C05485=1164.302,294.931,-71.199,-176.927,8.045,148.667
C05486=1164.298,295.179,-71.230,-176.924,8.049,148.668
C05487=1164.294,295.428,-71.259,-176.921,8.052,148.668
C05488=1164.290,295.675,-71.290,-176.919,8.055,148.668
C05489=1164.285,295.924,-71.320,-176.916,8.058,148.668
C05490=1164.282,296.172,-71.350,-176.914,8.061,148.668
C05491=1164.277,296.420,-71.381,-176.911,8.064,148.668
C05492=1164.273,296.668,-71.410,-176.909,8.067,148.668
C05493=1164.269,296.916,-71.441,-176.906,8.070,148.668
C05494=1164.265,297.164,-71.471,-176.904,8.073,148.668
C05495=1164.260,297.413,-71.501,-176.901,8.076,148.668
C05496=1164.256,297.660,-71.532,-176.898,8.079,148.668
C05497=1164.251,297.908,-71.562,-176.896,8.083,148.668
C05498=1164.247,298.157,-71.592,-176.893,8.086,148.668
C05499=1164.243,298.405,-71.623,-176.891,8.089,148.668
C05500=1164.239,298.653,-71.653,-176.888,8.092,148.668
C05501=1164.234,298.901,-71.683,-176.885,8.095,148.668
C05502=1164.231,299.149,-71.713,-176.883,8.098,148.668
C05503=1164.226,299.397,-71.744,-176.880,8.101,148.668
C05504=1164.223,299.645,-71.775,-176.878,8.104,148.669
C05505=1164.218,299.893,-71.805,-176.875,8.107,148.668
C05506=1164.213,300.142,-71.835,-176.872,8.110,148.668
C05507=1164.209,300.390,-71.866,-176.870,8.114,148.669
C05508=1164.205,300.638,-71.897,-176.867,8.117,148.669
C05509=1164.201,300.886,-71.927,-176.865,8.120,148.669
C05510=1164.197,301.134,-71.958,-176.862,8.123,148.669
C05511=1164.192,301.382,-71.988,-176.860,8.126,148.669
C05512=1164.189,301.630,-72.019,-176.857,8.130,148.669
C05513=1164.184,301.879,-72.049,-176.854,8.133,148.669
C05514=1164.179,302.127,-72.080,-176.852,8.136,148.669
C05515=1164.175,302.374,-72.110,-176.849,8.139,148.669
C05516=1164.171,302.623,-72.141,-176.847,8.142,148.669
C05517=1164.167,302.871,-72.172,-176.844,8.145,148.669
C05518=1164.163,303.119,-72.202,-176.841,8.148,148.669
C05519=1164.158,303.367,-72.233,-176.839,8.152,148.669
C05520=1164.154,303.615,-72.264,-176.836,8.155,148.669
C05521=1164.150,303.863,-72.295,-176.834,8.158,148.670
C05522=1164.146,304.111,-72.325,-176.831,8.161,148.670
C05523=1164.142,304.359,-72.356,-176.829,8.164,148.670
C05524=1164.137,304.607,-72.387,-176.826,8.167,148.670
C05525=1164.133,304.855,-72.417,-176.824,8.170,148.670
C05526=1164.130,305.103,-72.449,-176.821,8.173,148.670
C05527=1164.125,305.351,-72.479,-176.818,8.177,148.670
C05528=1164.120,305.599,-72.510,-176.815,8.180,148.670
C05529=1164.116,305.848,-72.541,-176.813,8.184,148.670
C05530=1164.113,306.095,-72.572,-176.810,8.187,148.670
C05531=1164.108,306.343,-72.602,-176.808,8.190,148.670
C05532=1164.104,306.592,-72.633,-176.805,8.193,148.670
C05533=1164.099,306.840,-72.664,-176.803,8.196,148.670
C05534=1164.095,307.087,-72.696,-176.800,8.199,148.671
C05535=1164.091,307.336,-72.727,-176.797,8.202,148.671
C05536=1164.087,307.584,-72.757,-176.795,8.205,148.671
C05537=1164.083,307.832,-72.788,-176.792,8.208,148.671
C05538=1164.079,308.080,-72.820,-176.790,8.212,148.671
C05539=1164.074,308.328,-72.850,-176.787,8.215,148.671
C05540=1164.070,308.576,-72.881,-176.785,8.219,148.671
C05541=1164.066,308.824,-72.912,-176.782,8.222,148.671
C05542=1164.062,309.072,-72.944,-176.780,8.225,148.671
C05543=1164.057,309.320,-72.975,-176.777,8.228,148.671
C05544=1164.053,309.568,-73.005,-176.774,8.231,148.671
C05545=1164.050,309.816,-73.037,-176.772,8.235,148.672
C05546=1164.045,310.064,-73.068,-176.769,8.238,148.672
C05547=1164.041,310.312,-73.099,-176.767,8.241,148.672
C05548=1164.037,310.560,-73.130,-176.764,8.244,148.672
C05549=1164.033,310.808,-73.161,-176.762,8.248,148.672
C05550=1164.028,311.056,-73.193,-176.759,8.251,148.672
C05551=1164.024,311.304,-73.224,-176.756,8.254,148.672
C05552=1164.020,311.552,-73.255,-176.754,8.257,148.672
C05553=1164.015,311.800,-73.286,-176.751,8.260,148.672
C05554=1164.011,312.048,-73.317,-176.749,8.263,148.672
C05555=1164.007,312.296,-73.349,-176.746,8.267,148.673
C05556=1164.003,312.544,-73.380,-176.744,8.270,148.672
C05557=1163.999,312.792,-73.411,-176.741,8.273,148.673
C05558=1163.995,313.040,-73.443,-176.738,8.277,148.673
C05559=1163.991,313.288,-73.474,-176.736,8.280,148.673
C05560=1163.986,313.565,-73.510,-176.733,8.283,148.673
C05561=1163.981,313.843,-73.544,-176.730,8.287,148.673
C05562=1163.976,314.119,-73.579,-176.728,8.290,148.673
C05563=1163.972,314.397,-73.615,-176.725,8.294,148.673
C05564=1163.967,314.644,-73.646,-176.722,8.298,148.674
C05565=1163.963,314.893,-73.678,-176.719,8.300,148.674
C05566=1163.959,315.140,-73.709,-176.717,8.304,148.674
C05567=1163.955,315.388,-73.741,-176.714,8.308,148.674
C05568=1163.951,315.636,-73.772,-176.712,8.311,148.674
C05569=1163.947,315.884,-73.804,-176.709,8.314,148.674
C05570=1163.943,316.132,-73.835,-176.707,8.317,148.674
C05571=1163.939,316.380,-73.866,-176.704,8.320,148.674
C05572=1163.934,316.629,-73.899,-176.702,8.324,148.674
C05573=1163.930,316.876,-73.930,-176.699,8.327,148.674
C05574=1163.926,317.124,-73.962,-176.696,8.331,148.675
C05575=1163.922,317.373,-73.993,-176.694,8.334,148.675
C05576=1163.918,317.620,-74.025,-176.691,8.337,148.675
C05577=1163.914,317.868,-74.057,-176.689,8.340,148.675
C05578=1163.909,318.116,-74.088,-176.686,8.343,148.675
C05579=1163.905,318.364,-74.120,-176.684,8.347,148.675
C05580=1163.902,318.612,-74.151,-176.682,8.350,148.675
C05581=1163.897,318.860,-74.183,-176.678,8.354,148.675
C05582=1163.893,319.108,-74.215,-176.676,8.357,148.676
C05583=1163.888,319.356,-74.247,-176.673,8.360,148.676
C05584=1163.885,319.604,-74.279,-176.671,8.363,148.676
C05585=1163.881,319.852,-74.311,-176.669,8.367,148.676
C05586=1163.876,320.099,-74.343,-176.666,8.369,148.676
C05587=1163.872,320.347,-74.374,-176.663,8.374,148.676
C05588=1163.868,320.596,-74.406,-176.661,8.377,148.676
C05589=1163.863,320.844,-74.438,-176.658,8.380,148.676
C05590=1163.860,321.092,-74.469,-176.656,8.383,148.677
C05591=1163.856,321.340,-74.501,-176.653,8.386,148.677
C05592=1163.852,321.587,-74.533,-176.651,8.389,148.677
C05593=1163.847,321.835,-74.565,-176.648,8.393,148.677
C05594=1163.843,322.083,-74.597,-176.646,8.397,148.677
C05595=1163.840,322.331,-74.629,-176.643,8.400,148.677
C05596=1163.835,322.578,-74.662,-176.640,8.403,148.677
C05597=1163.831,322.826,-74.694,-176.638,8.406,148.678
C05598=1163.827,323.075,-74.726,-176.635,8.409,148.678
C05599=1163.822,323.322,-74.757,-176.633,8.413,148.678
C05600=1163.819,323.570,-74.789,-176.630,8.417,148.678
C05601=1163.814,323.819,-74.822,-176.628,8.420,148.678
C05602=1163.811,324.067,-74.854,-176.625,8.423,148.678
C05603=1163.806,324.314,-74.886,-176.623,8.426,148.678
C05604=1163.802,324.562,-74.918,-176.621,8.430,148.679
C05605=1163.798,324.810,-74.950,-176.617,8.433,148.679
C05606=1163.794,325.058,-74.983,-176.615,8.437,148.679
C05607=1163.790,325.305,-75.014,-176.613,8.440,148.679
C05608=1163.785,325.554,-75.046,-176.610,8.443,148.679
C05609=1163.782,325.802,-75.078,-176.608,8.446,148.679
C05610=1163.777,326.050,-75.111,-176.605,8.450,148.680
C05611=1163.774,326.298,-75.143,-176.603,8.454,148.680
C05612=1163.769,326.545,-75.175,-176.600,8.457,148.680
C05613=1163.765,326.793,-75.208,-176.598,8.460,148.680
C05614=1163.761,327.041,-75.240,-176.595,8.463,148.680
C05615=1163.757,327.289,-75.272,-176.592,8.467,148.680
C05616=1163.753,327.537,-75.305,-176.590,8.470,148.680
C05617=1163.749,327.784,-75.337,-176.587,8.474,148.681
C05618=1163.744,328.032,-75.369,-176.585,8.477,148.681
C05619=1163.740,328.280,-75.402,-176.583,8.480,148.681
C05620=1163.736,328.528,-75.434,-176.579,8.484,148.681
C05621=1163.732,328.777,-75.467,-176.577,8.487,148.681
C05622=1163.728,329.023,-75.499,-176.575,8.490,148.681
C05623=1163.724,329.272,-75.531,-176.573,8.494,148.682
C05624=1163.720,329.519,-75.564,-176.570,8.497,148.682
C05625=1163.716,329.767,-75.596,-176.567,8.501,148.682
C05626=1163.711,330.016,-75.629,-176.565,8.504,148.682
C05627=1163.708,330.263,-75.661,-176.562,8.507,148.682
C05628=1163.703,330.512,-75.694,-176.560,8.511,148.682
C05629=1163.699,330.759,-75.727,-176.558,8.514,148.683
C05630=1163.695,331.007,-75.758,-176.554,8.518,148.683
C05631=1163.691,331.254,-75.792,-176.552,8.521,148.683
C05632=1163.687,331.502,-75.825,-176.550,8.524,148.683
C05633=1163.683,331.750,-75.857,-176.548,8.528,148.683
C05634=1163.679,331.998,-75.890,-176.545,8.532,148.684
C05635=1163.674,332.246,-75.922,-176.542,8.535,148.684
C05636=1163.670,332.494,-75.955,-176.540,8.538,148.684
C05637=1163.667,332.741,-75.988,-176.537,8.541,148.684
C05638=1163.662,332.990,-76.020,-176.534,8.545,148.684
C05639=1163.658,333.237,-76.054,-176.532,8.549,148.684
C05640=1163.654,333.485,-76.085,-176.530,8.552,148.685
C05641=1163.650,333.732,-76.118,-176.527,8.555,148.685
C05642=1163.646,333.980,-76.151,-176.524,8.559,148.685
C05643=1163.642,334.228,-76.184,-176.522,8.562,148.685
C05644=1163.637,334.476,-76.217,-176.520,8.566,148.685
C05645=1163.634,334.724,-76.249,-176.517,8.569,148.685
C05646=1163.630,334.971,-76.283,-176.515,8.572,148.686
C05647=1163.625,335.220,-76.315,-176.512,8.576,148.686
C05648=1163.621,335.467,-76.348,-176.509,8.579,148.686
C05649=1163.617,335.715,-76.381,-176.507,8.583,148.686
C05650=1163.613,335.963,-76.414,-176.505,8.586,148.686
C05651=1163.609,336.210,-76.447,-176.502,8.590,148.687
C05652=1163.605,336.459,-76.480,-176.500,8.593,148.687
C05653=1163.601,336.706,-76.513,-176.497,8.597,148.687
C05654=1163.597,336.954,-76.546,-176.494,8.601,148.687
C05655=1163.592,337.202,-76.579,-176.492,8.604,148.687
C05656=1163.588,337.450,-76.612,-176.490,8.607,148.688
C05657=1163.585,337.697,-76.645,-176.487,8.610,148.688
C05658=1163.581,337.945,-76.678,-176.484,8.614,148.688
C05659=1163.577,338.192,-76.711,-176.482,8.618,148.688
C05660=1163.572,338.440,-76.744,-176.480,8.621,148.688
C05661=1163.568,338.688,-76.777,-176.477,8.624,148.688
C05662=1163.564,338.936,-76.811,-176.475,8.628,148.689
C05663=1163.560,339.183,-76.844,-176.472,8.632,148.689
C05664=1163.555,339.464,-76.880,-176.469,8.636,148.689
C05665=1163.551,339.743,-76.918,-176.466,8.640,148.689
C05666=1163.546,340.023,-76.956,-176.464,8.643,148.690
C05667=1163.541,340.302,-76.993,-176.461,8.647,148.690
C05668=1163.538,340.551,-77.027,-176.458,8.651,148.690
C05669=1163.534,340.799,-77.060,-176.456,8.655,148.690
C05670=1163.530,341.046,-77.093,-176.454,8.658,148.691
C05671=1163.525,341.294,-77.126,-176.452,8.661,148.691
C05672=1163.522,341.541,-77.160,-176.449,8.665,148.691
C05673=1163.517,341.789,-77.193,-176.446,8.669,148.691
C05674=1163.513,342.037,-77.226,-176.444,8.672,148.691
C05675=1163.509,342.284,-77.259,-176.441,8.676,148.692
C05676=1163.505,342.532,-77.293,-176.439,8.679,148.692
C05677=1163.501,342.780,-77.326,-176.437,8.683,148.692
C05678=1163.497,343.028,-77.361,-176.434,8.687,148.692
C05679=1163.493,343.276,-77.394,-176.431,8.690,148.693
C05680=1163.489,343.523,-77.427,-176.429,8.693,148.693
C05681=1163.484,343.771,-77.460,-176.427,8.697,148.693
C05682=1163.480,344.019,-77.493,-176.424,8.701,148.693
C05683=1163.477,344.266,-77.527,-176.422,8.704,148.693
C05684=1163.472,344.514,-77.560,-176.419,8.707,148.694
C05685=1163.469,344.762,-77.594,-176.417,8.711,148.694
C05686=1163.464,345.009,-77.628,-176.414,8.715,148.694
C05687=1163.460,345.257,-77.661,-176.412,8.718,148.694
C05688=1163.456,345.505,-77.694,-176.409,8.722,148.695
C05689=1163.452,345.752,-77.728,-176.407,8.725,148.695
C05690=1163.448,346.000,-77.762,-176.404,8.729,148.695
C05691=1163.444,346.249,-77.796,-176.402,8.733,148.695
C05692=1163.440,346.496,-77.830,-176.399,8.736,148.696
C05693=1163.436,346.743,-77.863,-176.397,8.739,148.696
C05694=1163.432,346.990,-77.897,-176.394,8.744,148.696
C05695=1163.428,347.239,-77.931,-176.392,8.747,148.696
C05696=1163.424,347.487,-77.964,-176.390,8.750,148.696
C05697=1163.420,347.734,-77.998,-176.387,8.754,148.697
C05698=1163.416,347.982,-78.031,-176.385,8.758,148.697
C05699=1163.411,348.229,-78.065,-176.382,8.761,148.697
C05700=1163.407,348.478,-78.099,-176.380,8.765,148.698
C05701=1163.404,348.725,-78.133,-176.377,8.769,148.698
C05702=1163.399,348.972,-78.166,-176.375,8.772,148.698
C05703=1163.395,349.220,-78.200,-176.372,8.776,148.698
C05704=1163.392,349.468,-78.235,-176.370,8.779,148.698
C05705=1163.388,349.715,-78.268,-176.368,8.783,148.699
C05706=1163.383,349.963,-78.302,-176.365,8.787,148.699
C05707=1163.379,350.211,-78.336,-176.363,8.790,148.699
C05708=1163.376,350.458,-78.370,-176.361,8.794,148.700
C05709=1163.371,350.706,-78.404,-176.358,8.798,148.700
C05710=1163.367,350.954,-78.437,-176.355,8.801,148.700
C05711=1163.363,351.202,-78.472,-176.352,8.805,148.700
C05712=1163.359,351.449,-78.506,-176.350,8.808,148.701
C05713=1163.355,351.696,-78.539,-176.348,8.812,148.701
C05714=1163.351,351.945,-78.574,-176.345,8.816,148.701
C05715=1163.347,352.192,-78.608,-176.343,8.819,148.701
C05716=1163.342,352.440,-78.641,-176.341,8.823,148.702
C05717=1163.339,352.688,-78.676,-176.338,8.827,148.702
C05718=1163.335,352.935,-78.710,-176.336,8.830,148.702
C05719=1163.331,353.182,-78.744,-176.333,8.834,148.703
C05720=1163.327,353.430,-78.778,-176.331,8.838,148.703
C05721=1163.323,353.678,-78.812,-176.329,8.841,148.703
C05722=1163.319,353.926,-78.846,-176.326,8.845,148.703
C05723=1163.315,354.173,-78.881,-176.324,8.849,148.704
C05724=1163.311,354.420,-78.915,-176.322,8.852,148.704
C05725=1163.307,354.668,-78.949,-176.319,8.856,148.704
C05726=1163.303,354.915,-78.983,-176.316,8.859,148.704
C05727=1163.298,355.164,-79.017,-176.314,8.864,148.705
C05728=1163.295,355.411,-79.051,-176.312,8.867,148.705
C05729=1163.290,355.659,-79.086,-176.309,8.870,148.705
C05730=1163.287,355.907,-79.120,-176.307,8.875,148.706
C05731=1163.283,356.154,-79.154,-176.305,8.878,148.706
C05732=1163.279,356.402,-79.189,-176.302,8.882,148.706
C05733=1163.275,356.649,-79.223,-176.299,8.886,148.706
C05734=1163.271,356.896,-79.257,-176.297,8.889,148.707
C05735=1163.267,357.144,-79.292,-176.295,8.893,148.707
C05736=1163.262,357.392,-79.326,-176.292,8.897,148.707
C05737=1163.259,357.640,-79.361,-176.290,8.901,148.708
C05738=1163.255,357.887,-79.395,-176.288,8.904,148.708
C05739=1163.251,358.135,-79.429,-176.285,8.908,148.708
C05740=1163.247,358.382,-79.464,-176.283,8.912,148.709
C05741=1163.243,358.630,-79.499,-176.281,8.915,148.709
C05742=1163.239,358.877,-79.533,-176.278,8.919,148.709
C05743=1163.235,359.125,-79.568,-176.275,8.923,148.709
C05744=1163.231,359.372,-79.602,-176.273,8.927,148.710
C05745=1163.228,359.620,-79.637,-176.271,8.930,148.710
C05746=1163.223,359.868,-79.671,-176.268,8.934,148.710
C05747=1163.219,360.116,-79.706,-176.266,8.938,148.711
C05748=1163.215,360.363,-79.740,-176.263,8.942,148.711
C05749=1163.212,360.610,-79.775,-176.261,8.945,148.711
C05750=1163.207,360.858,-79.810,-176.258,8.950,148.712
C05751=1163.204,361.106,-79.844,-176.256,8.953,148.712
C05752=1163.199,361.353,-79.879,-176.254,8.958,148.712
C05753=1163.196,361.601,-79.914,-176.251,8.961,148.713
C05754=1163.191,361.848,-79.949,-176.249,8.964,148.713
C05755=1163.188,362.096,-79.983,-176.247,8.969,148.713
C05756=1163.183,362.343,-80.018,-176.244,8.972,148.714
C05757=1163.180,362.591,-80.053,-176.242,8.976,148.714
C05758=1163.176,362.839,-80.088,-176.240,8.980,148.714
C05759=1163.172,363.085,-80.122,-176.237,8.984,148.715
C05760=1163.168,363.333,-80.157,-176.235,8.987,148.715
C05761=1163.163,363.581,-80.192,-176.232,8.992,148.715
C05762=1163.160,363.828,-80.227,-176.230,8.995,148.716
C05763=1163.156,364.077,-80.262,-176.228,8.999,148.716
C05764=1163.152,364.324,-80.296,-176.226,9.003,148.717
C05765=1163.148,364.571,-80.331,-176.224,9.006,148.717
C05766=1163.144,364.819,-80.366,-176.221,9.011,148.717
C05767=1163.140,365.066,-80.401,-176.219,9.014,148.717
C05768=1163.136,365.348,-80.441,-176.216,9.018,148.718
C05769=1163.132,365.631,-80.481,-176.214,9.023,148.718
C05770=1163.127,365.913,-80.521,-176.211,9.028,148.719
C05771=1163.122,366.196,-80.561,-176.208,9.033,148.719
C05772=1163.118,366.444,-80.596,-176.206,9.036,148.720
C05773=1163.114,366.691,-80.631,-176.204,9.039,148.720
C05774=1163.110,366.939,-80.666,-176.202,9.044,148.721
C05775=1163.106,367.186,-80.702,-176.200,9.047,148.721
C05776=1163.102,367.434,-80.736,-176.197,9.052,148.721
C05777=1163.098,367.681,-80.772,-176.195,9.055,148.722
C05778=1163.095,367.929,-80.807,-176.193,9.059,148.722
C05779=1163.090,368.176,-80.842,-176.191,9.063,148.723
C05780=1163.086,368.424,-80.877,-176.189,9.067,148.723
C05781=1163.082,368.672,-80.912,-176.187,9.070,148.723
C05782=1163.078,368.919,-80.947,-176.185,9.075,148.724
C05783=1163.074,369.166,-80.983,-176.183,9.078,148.724
C05784=1163.071,369.414,-81.018,-176.181,9.082,148.725
C05785=1163.066,369.661,-81.053,-176.179,9.086,148.725
C05786=1163.062,369.908,-81.088,-176.177,9.090,148.726
C05787=1163.059,370.156,-81.124,-176.175,9.094,148.726
C05788=1163.055,370.404,-81.159,-176.172,9.098,148.727
C05789=1163.051,370.651,-81.194,-176.171,9.102,148.727
C05790=1163.047,370.898,-81.229,-176.169,9.106,148.728
C05791=1163.043,371.146,-81.265,-176.167,9.109,148.728
C05792=1163.039,371.393,-81.300,-176.165,9.114,148.729
C05793=1163.035,371.641,-81.335,-176.163,9.117,148.729
C05794=1163.031,371.888,-81.371,-176.161,9.121,148.730
C05795=1163.028,372.136,-81.406,-176.160,9.125,148.730
C05796=1163.023,372.383,-81.441,-176.157,9.129,148.730
C05797=1163.020,372.630,-81.477,-176.156,9.133,148.731
C05798=1163.016,372.878,-81.512,-176.154,9.137,148.732
C05799=1163.012,373.125,-81.549,-176.152,9.140,148.732
C05800=1163.008,373.373,-81.584,-176.151,9.144,148.733
C05801=1163.003,373.620,-81.619,-176.149,9.148,148.733
C05802=1163.000,373.868,-81.654,-176.147,9.152,148.734
C05803=1162.996,374.115,-81.690,-176.146,9.155,148.734
C05804=1162.992,374.363,-81.725,-176.143,9.160,148.735
C05805=1162.987,374.610,-81.761,-176.142,9.164,148.735
C05806=1162.984,374.857,-81.797,-176.140,9.167,148.736
C05807=1162.980,375.105,-81.832,-176.139,9.171,148.736
C05808=1162.977,375.352,-81.868,-176.137,9.175,148.737
C05809=1162.973,375.600,-81.903,-176.136,9.179,148.738
C05810=1162.969,375.847,-81.939,-176.134,9.183,148.738
C05811=1162.964,376.095,-81.975,-176.132,9.187,148.739
C05812=1162.961,376.342,-82.010,-176.131,9.190,148.739
C05813=1162.957,376.589,-82.046,-176.130,9.194,148.740
C05814=1162.953,376.836,-82.082,-176.129,9.197,148.741
C05815=1162.949,377.084,-82.118,-176.127,9.201,148.741
C05816=1162.945,377.332,-82.154,-176.126,9.205,148.742
C05817=1162.941,377.579,-82.189,-176.124,9.209,148.742
C05818=1162.938,377.826,-82.224,-176.123,9.213,148.743
C05819=1162.933,378.074,-82.260,-176.122,9.217,148.744
C05820=1162.929,378.321,-82.296,-176.121,9.220,148.744
C05821=1162.926,378.569,-82.332,-176.119,9.224,148.745
C05822=1162.922,378.816,-82.368,-176.118,9.228,148.745
C05823=1162.918,379.064,-82.404,-176.117,9.232,148.746
C05824=1162.914,379.310,-82.439,-176.116,9.235,148.747
C05825=1162.909,379.558,-82.475,-176.114,9.239,148.747
C05826=1162.906,379.806,-82.511,-176.113,9.243,148.748
C05827=1162.902,380.053,-82.547,-176.113,9.246,148.749
C05828=1162.899,380.300,-82.583,-176.111,9.250,148.750
C05829=1162.894,380.548,-82.619,-176.111,9.254,148.750
C05830=1162.891,380.795,-82.654,-176.109,9.258,148.751
C05831=1162.887,381.043,-82.691,-176.108,9.261,148.751
C05832=1162.882,381.289,-82.726,-176.107,9.265,148.752
C05833=1162.879,381.537,-82.762,-176.107,9.268,148.753
C05834=1162.874,381.785,-82.798,-176.106,9.272,148.754
C05835=1162.871,382.032,-82.834,-176.105,9.276,148.754
C05836=1162.867,382.279,-82.870,-176.104,9.279,148.755
C05837=1162.863,382.527,-82.906,-176.103,9.283,148.756
C05838=1162.859,382.774,-82.942,-176.103,9.286,148.757
C05839=1162.855,383.022,-82.978,-176.102,9.289,148.757
C05840=1162.851,383.269,-83.014,-176.101,9.293,148.758
C05841=1162.848,383.516,-83.050,-176.100,9.297,148.759
C05842=1162.844,383.764,-83.086,-176.100,9.300,148.760
C05843=1162.840,384.011,-83.122,-176.099,9.303,148.760
C05844=1162.836,384.258,-83.159,-176.099,9.307,148.761
C05845=1162.832,384.506,-83.194,-176.098,9.311,148.762
C05846=1162.828,384.753,-83.230,-176.097,9.314,148.762
C05847=1162.824,385.000,-83.266,-176.097,9.318,148.763
C05848=1162.820,385.247,-83.302,-176.096,9.321,148.764
C05849=1162.816,385.495,-83.339,-176.096,9.325,148.765
C05850=1162.812,385.742,-83.374,-176.096,9.328,148.766
C05851=1162.808,385.990,-83.410,-176.096,9.330,148.766
C05852=1162.805,386.237,-83.447,-176.095,9.334,148.767
C05853=1162.800,386.485,-83.483,-176.095,9.337,148.768
C05854=1162.797,386.731,-83.519,-176.094,9.341,148.769
C05855=1162.793,386.979,-83.555,-176.094,9.344,148.769
C05856=1162.789,387.226,-83.592,-176.094,9.347,148.770
C05857=1162.785,387.474,-83.627,-176.094,9.350,148.771
C05858=1162.781,387.721,-83.664,-176.094,9.354,148.772
C05859=1162.778,387.968,-83.699,-176.094,9.356,148.772
C05860=1162.774,388.216,-83.736,-176.094,9.360,148.773
C05861=1162.770,388.463,-83.772,-176.094,9.362,148.774
C05862=1162.766,388.710,-83.809,-176.093,9.366,148.775
C05863=1162.762,388.958,-83.844,-176.094,9.368,148.776
C05864=1162.758,389.205,-83.881,-176.094,9.372,148.777
C05865=1162.754,389.452,-83.917,-176.094,9.375,148.777
C05866=1162.750,389.700,-83.954,-176.094,9.377,148.778
C05867=1162.747,389.947,-83.989,-176.094,9.381,148.779
C05868=1162.743,390.194,-84.026,-176.094,9.384,148.780
C05869=1162.739,390.442,-84.062,-176.094,9.386,148.780
C05870=1162.735,390.689,-84.098,-176.094,9.390,148.781
C05871=1162.731,390.937,-84.134,-176.094,9.392,148.782
C05872=1162.726,391.222,-84.177,-176.095,9.395,148.783
C05873=1162.722,391.508,-84.218,-176.095,9.399,148.784
C05874=1162.718,391.793,-84.260,-176.095,9.402,148.785
C05875=1162.713,392.078,-84.302,-176.095,9.406,148.786
C05876=1162.709,392.325,-84.338,-176.095,9.408,148.787
C05877=1162.705,392.574,-84.375,-176.096,9.411,148.787
C05878=1162.702,392.820,-84.411,-176.096,9.414,148.788
C05879=1162.698,393.068,-84.447,-176.096,9.416,148.789
C05880=1162.694,393.315,-84.483,-176.097,9.419,148.790
C05881=1162.690,393.562,-84.520,-176.097,9.422,148.790
C05882=1162.687,393.810,-84.556,-176.097,9.424,148.791
C05883=1162.683,394.057,-84.592,-176.098,9.427,148.792
C05884=1162.678,394.305,-84.629,-176.098,9.429,148.793
C05885=1162.675,394.552,-84.665,-176.099,9.432,148.794
C05886=1162.671,394.799,-84.702,-176.099,9.434,148.794
C05887=1162.667,395.046,-84.737,-176.100,9.437,148.795
C05888=1162.663,395.294,-84.774,-176.100,9.440,148.796
C05889=1162.659,395.541,-84.810,-176.100,9.441,148.797
C05890=1162.655,395.788,-84.847,-176.101,9.444,148.798
C05891=1162.651,396.035,-84.883,-176.101,9.447,148.798
C05892=1162.647,396.283,-84.919,-176.101,9.449,148.799
C05893=1162.643,396.530,-84.956,-176.102,9.451,148.800
C05894=1162.640,396.778,-84.991,-176.103,9.454,148.801
C05895=1162.636,397.025,-85.028,-176.104,9.456,148.801
C05896=1162.632,397.272,-85.064,-176.104,9.459,148.802
C05897=1162.628,397.520,-85.101,-176.104,9.461,148.803
C05898=1162.624,397.767,-85.137,-176.105,9.463,148.804
C05899=1162.620,398.014,-85.174,-176.105,9.466,148.804
C05900=1162.616,398.261,-85.210,-176.106,9.468,148.805
C05901=1162.613,398.508,-85.246,-176.107,9.470,148.806
C05902=1162.608,398.755,-85.283,-176.107,9.472,148.807
C05903=1162.604,399.003,-85.319,-176.107,9.475,148.807
C05904=1162.601,399.250,-85.355,-176.108,9.477,148.808
C05905=1162.597,399.497,-85.392,-176.109,9.479,148.809
C05906=1162.593,399.745,-85.428,-176.109,9.481,148.809
C05907=1162.589,399.992,-85.465,-176.109,9.484,148.810
C05908=1162.585,400.239,-85.502,-176.111,9.486,148.811
C05909=1162.581,400.487,-85.537,-176.111,9.488,148.812
C05910=1162.578,400.735,-85.574,-176.111,9.490,148.812
C05911=1162.574,400.982,-85.611,-176.112,9.493,148.813
C05912=1162.570,401.229,-85.647,-176.113,9.495,148.814
C05913=1162.566,401.477,-85.684,-176.113,9.496,148.815
C05914=1162.562,401.723,-85.720,-176.114,9.499,148.815
C05915=1162.558,401.971,-85.756,-176.114,9.501,148.816
C05916=1162.555,402.218,-85.792,-176.115,9.502,148.817
C05917=1162.551,402.465,-85.829,-176.115,9.505,148.817
C05918=1162.546,402.713,-85.865,-176.116,9.507,148.818
C05919=1162.543,402.960,-85.902,-176.117,9.509,148.819
C05920=1162.539,403.207,-85.938,-176.117,9.511,148.819
C05921=1162.535,403.455,-85.974,-176.118,9.513,148.820
C05922=1162.531,403.702,-86.011,-176.118,9.515,148.821
C05923=1162.527,403.949,-86.048,-176.119,9.517,148.821
C05924=1162.523,404.197,-86.083,-176.120,9.520,148.822
C05925=1162.519,404.444,-86.120,-176.120,9.521,148.823
C05926=1162.515,404.691,-86.157,-176.121,9.523,148.824
C05927=1162.512,404.938,-86.193,-176.122,9.525,148.824
C05928=1162.508,405.186,-86.230,-176.122,9.527,148.825
C05929=1162.504,405.433,-86.266,-176.123,9.529,148.826
C05930=1162.500,405.680,-86.303,-176.123,9.531,148.826
C05931=1162.496,405.928,-86.339,-176.124,9.533,148.827
C05932=1162.493,406.175,-86.375,-176.124,9.535,148.828
C05933=1162.489,406.422,-86.412,-176.125,9.537,148.828
C05934=1162.484,406.669,-86.449,-176.126,9.539,148.829
C05935=1162.481,406.917,-86.484,-176.126,9.540,148.830
C05936=1162.477,407.164,-86.521,-176.127,9.542,148.830
C05937=1162.473,407.411,-86.558,-176.127,9.545,148.831
C05938=1162.469,407.659,-86.594,-176.128,9.546,148.832
C05939=1162.465,407.906,-86.631,-176.129,9.548,148.832
C05940=1162.461,408.153,-86.667,-176.129,9.550,148.833
C05941=1162.457,408.400,-86.704,-176.129,9.551,148.833
C05942=1162.453,408.648,-86.740,-176.130,9.554,148.834
C05943=1162.450,408.895,-86.776,-176.130,9.556,148.835
C05944=1162.446,409.143,-86.813,-176.131,9.557,148.835
C05945=1162.442,409.390,-86.849,-176.132,9.559,148.836
C05946=1162.438,409.637,-86.886,-176.132,9.561,148.837
C05947=1162.434,409.885,-86.923,-176.133,9.562,148.837
C05948=1162.430,410.132,-86.959,-176.133,9.565,148.838
C05949=1162.427,410.379,-86.995,-176.134,9.567,148.838
C05950=1162.422,410.626,-87.032,-176.134,9.568,148.839
C05951=1162.419,410.873,-87.068,-176.135,9.570,148.840
C05952=1162.415,411.121,-87.105,-176.135,9.572,148.840
C05953=1162.411,411.368,-87.141,-176.136,9.573,148.841
C05954=1162.407,411.615,-87.177,-176.137,9.575,148.841
C05955=1162.403,411.862,-87.214,-176.137,9.578,148.842
C05956=1162.399,412.110,-87.251,-176.137,9.579,148.843
C05957=1162.396,412.358,-87.287,-176.138,9.581,148.843
C05958=1162.392,412.605,-87.324,-176.138,9.583,148.844
C05959=1162.388,412.852,-87.361,-176.139,9.584,148.845
C05960=1162.384,413.099,-87.397,-176.139,9.586,148.845
C05961=1162.380,413.347,-87.433,-176.139,9.588,148.846
C05962=1162.376,413.594,-87.470,-176.140,9.590,148.846
C05963=1162.373,413.841,-87.506,-176.140,9.592,148.847
C05964=1162.368,414.088,-87.543,-176.141,9.593,148.847
C05965=1162.364,414.335,-87.580,-176.142,9.595,148.848
C05966=1162.361,414.583,-87.616,-176.142,9.596,148.849
C05967=1162.357,414.830,-87.652,-176.142,9.599,148.849
C05968=1162.353,415.077,-87.689,-176.142,9.600,148.850
C05969=1162.350,415.325,-87.726,-176.143,9.602,148.850
C05970=1162.347,415.572,-87.762,-176.144,9.604,148.851
C05971=1162.345,415.820,-87.799,-176.144,9.605,148.851
C05972=1162.345,416.166,-87.850,-176.145,9.608,148.852
C05973=1162.346,416.512,-87.899,-176.145,9.610,148.853
C05974=1162.348,416.857,-87.950,-176.146,9.613,148.854
C05975=1162.352,417.203,-88.000,-176.146,9.614,148.854
C05976=1161.932,417.205,-88.046,-176.149,9.625,148.858
C05977=1161.927,416.856,-87.995,-176.149,9.624,148.857
C05978=1161.924,416.507,-87.945,-176.148,9.621,148.857
C05979=1161.923,416.158,-87.894,-176.147,9.619,148.856
C05980=1161.924,415.809,-87.843,-176.147,9.616,148.855
C05981=1161.926,415.561,-87.807,-176.147,9.615,148.855
C05982=1161.929,415.314,-87.770,-176.146,9.613,148.854
C05983=1161.931,415.066,-87.733,-176.146,9.611,148.853
C05984=1161.936,414.819,-87.697,-176.145,9.610,148.853
C05985=1161.940,414.571,-87.660,-176.145,9.607,148.852
C05986=1161.943,414.324,-87.624,-176.145,9.606,148.852
C05987=1161.947,414.077,-87.587,-176.144,9.604,148.851
C05988=1161.952,413.830,-87.550,-176.144,9.603,148.851
C05989=1161.955,413.582,-87.515,-176.143,9.601,148.850
C05990=1161.959,413.335,-87.478,-176.142,9.599,148.849
C05991=1161.963,413.088,-87.441,-176.142,9.598,148.849
C05992=1161.967,412.841,-87.405,-176.142,9.595,148.848
C05993=1161.971,412.593,-87.369,-176.141,9.593,148.847
C05994=1161.975,412.346,-87.332,-176.140,9.592,148.847
C05995=1161.978,412.098,-87.295,-176.140,9.590,148.846
C05996=1161.982,411.851,-87.258,-176.139,9.588,148.846
C05997=1161.986,411.604,-87.222,-176.139,9.587,148.845
C05998=1161.990,411.357,-87.186,-176.139,9.584,148.844
C05999=1161.994,411.109,-87.149,-176.138,9.583,148.844
C06000=1161.998,410.862,-87.112,-176.138,9.581,148.843
C06001=1162.001,410.615,-87.076,-176.137,9.579,148.843
C06002=1162.006,410.368,-87.040,-176.136,9.577,148.842
C06003=1162.010,410.120,-87.003,-176.136,9.576,148.841
C06004=1162.013,409.873,-86.967,-176.135,9.574,148.841
C06005=1162.017,409.626,-86.930,-176.135,9.572,148.840
C06006=1162.022,409.378,-86.894,-176.134,9.570,148.840
C06007=1162.025,409.132,-86.857,-176.134,9.568,148.839
C06008=1162.029,408.884,-86.820,-176.133,9.566,148.838
C06009=1162.033,408.636,-86.783,-176.132,9.565,148.838
C06010=1162.036,408.389,-86.748,-176.132,9.563,148.837
C06011=1162.040,408.142,-86.711,-176.132,9.560,148.836
C06012=1162.044,407.895,-86.675,-176.131,9.559,148.836
C06013=1162.048,407.648,-86.638,-176.131,9.557,148.835
C06014=1162.052,407.400,-86.602,-176.130,9.555,148.835
C06015=1162.056,407.153,-86.565,-176.129,9.554,148.834
C06016=1162.060,406.906,-86.529,-176.128,9.552,148.833
C06017=1162.064,406.658,-86.492,-176.128,9.549,148.832
C06018=1162.067,406.411,-86.456,-176.128,9.548,148.832
C06019=1162.072,406.164,-86.419,-176.127,9.546,148.831
C06020=1162.076,405.917,-86.382,-176.126,9.544,148.831
C06021=1162.079,405.669,-86.347,-176.126,9.542,148.830
C06022=1162.083,405.421,-86.310,-176.125,9.540,148.829
C06023=1162.086,405.174,-86.273,-176.125,9.538,148.829
C06024=1162.091,404.927,-86.237,-176.124,9.536,148.828
C06025=1162.095,404.679,-86.200,-176.123,9.535,148.827
C06026=1162.098,404.433,-86.164,-176.123,9.532,148.826
C06027=1162.102,404.185,-86.127,-176.122,9.530,148.826
C06028=1162.107,403.938,-86.091,-176.121,9.528,148.825
C06029=1162.110,403.691,-86.055,-176.121,9.526,148.824
C06030=1162.114,403.444,-86.018,-176.121,9.524,148.824
C06031=1162.118,403.196,-85.982,-176.120,9.522,148.823
C06032=1162.122,402.949,-85.946,-176.119,9.520,148.822
C06033=1162.126,402.702,-85.909,-176.118,9.519,148.822
C06034=1162.129,402.455,-85.873,-176.118,9.516,148.821
C06035=1162.134,402.207,-85.836,-176.117,9.514,148.820
C06036=1162.138,401.960,-85.800,-176.116,9.512,148.820
C06037=1162.141,401.713,-85.763,-176.116,9.510,148.819
C06038=1162.145,401.464,-85.727,-176.116,9.508,148.818
C06039=1162.148,401.218,-85.690,-176.114,9.506,148.817
C06040=1162.152,400.970,-85.654,-176.114,9.503,148.817
C06041=1162.157,400.723,-85.617,-176.114,9.502,148.816
C06042=1162.160,400.476,-85.581,-176.114,9.499,148.815
C06043=1162.164,400.228,-85.544,-176.112,9.497,148.814
C06044=1162.169,399.981,-85.508,-176.112,9.495,148.814
C06045=1162.172,399.734,-85.472,-176.112,9.493,148.813
C06046=1162.176,399.487,-85.435,-176.110,9.491,148.812
C06047=1162.180,399.239,-85.400,-176.110,9.488,148.812
C06048=1162.184,398.992,-85.363,-176.110,9.486,148.811
C06049=1162.188,398.745,-85.326,-176.109,9.483,148.810
C06050=1162.191,398.497,-85.290,-176.108,9.482,148.809
C06051=1162.196,398.250,-85.253,-176.108,9.479,148.809
C06052=1162.199,398.003,-85.217,-176.107,9.477,148.808
C06053=1162.203,397.755,-85.181,-176.107,9.474,148.807
C06054=1162.207,397.508,-85.144,-176.106,9.473,148.806
C06055=1162.211,397.261,-85.108,-176.106,9.470,148.805
C06056=1162.215,397.013,-85.072,-176.106,9.467,148.805
C06057=1162.219,396.767,-85.035,-176.104,9.465,148.804
C06058=1162.223,396.519,-84.999,-176.104,9.463,148.803
C06059=1162.227,396.272,-84.962,-176.104,9.460,148.803
C06060=1162.230,396.024,-84.926,-176.103,9.458,148.802
C06061=1162.234,395.777,-84.889,-176.103,9.455,148.801
C06062=1162.238,395.529,-84.853,-176.102,9.453,148.800
C06063=1162.242,395.282,-84.817,-176.102,9.451,148.799
C06064=1162.245,395.035,-84.781,-176.101,9.448,148.799
C06065=1162.249,394.787,-84.744,-176.101,9.445,148.798
C06066=1162.254,394.540,-84.707,-176.101,9.443,148.797
C06067=1162.257,394.293,-84.672,-176.100,9.440,148.796
C06068=1162.261,394.045,-84.635,-176.100,9.438,148.796
C06069=1162.265,393.799,-84.599,-176.099,9.435,148.795
C06070=1162.269,393.551,-84.563,-176.099,9.433,148.794
C06071=1162.272,393.304,-84.526,-176.099,9.430,148.793
C06072=1162.277,393.056,-84.490,-176.098,9.427,148.792
C06073=1162.280,392.809,-84.454,-176.098,9.425,148.792
C06074=1162.284,392.562,-84.417,-176.097,9.422,148.791
C06075=1162.289,392.314,-84.381,-176.097,9.419,148.790
C06076=1162.292,392.067,-84.345,-176.097,9.416,148.789
C06077=1162.296,391.782,-84.303,-176.097,9.413,148.788
C06078=1162.301,391.496,-84.260,-176.097,9.410,148.787
C06079=1162.305,391.210,-84.219,-176.096,9.407,148.786
C06080=1162.310,390.924,-84.177,-176.096,9.404,148.786
C06081=1162.314,390.678,-84.141,-176.095,9.401,148.785
C06082=1162.318,390.430,-84.104,-176.095,9.398,148.784
C06083=1162.321,390.183,-84.068,-176.096,9.395,148.783
C06084=1162.325,389.936,-84.032,-176.095,9.392,148.782
C06085=1162.329,389.688,-83.996,-176.095,9.389,148.782
C06086=1162.333,389.441,-83.959,-176.096,9.386,148.781
C06087=1162.337,389.193,-83.924,-176.095,9.383,148.780
C06088=1162.341,388.946,-83.887,-176.095,9.380,148.779
C06089=1162.345,388.699,-83.851,-176.095,9.377,148.778
C06090=1162.349,388.452,-83.814,-176.095,9.374,148.777
C06091=1162.352,388.204,-83.779,-176.095,9.371,148.777
C06092=1162.356,387.957,-83.742,-176.095,9.368,148.776
C06093=1162.360,387.709,-83.706,-176.095,9.365,148.775
C06094=1162.364,387.462,-83.670,-176.095,9.361,148.774
C06095=1162.368,387.215,-83.634,-176.095,9.359,148.774
C06096=1162.372,386.967,-83.597,-176.096,9.355,148.773
C06097=1162.376,386.720,-83.562,-176.096,9.352,148.772
C06098=1162.380,386.474,-83.526,-176.097,9.348,148.771
C06099=1162.384,386.226,-83.490,-176.097,9.346,148.771
C06100=1162.387,385.979,-83.453,-176.097,9.342,148.770
C06101=1162.392,385.731,-83.417,-176.097,9.339,148.769
C06102=1162.395,385.484,-83.381,-176.097,9.335,148.768
C06103=1162.400,385.237,-83.345,-176.098,9.332,148.767
C06104=1162.403,384.989,-83.309,-176.098,9.329,148.767
C06105=1162.407,384.742,-83.272,-176.099,9.325,148.766
C06106=1162.411,384.494,-83.237,-176.100,9.322,148.765
C06107=1162.415,384.247,-83.200,-176.100,9.319,148.764
C06108=1162.419,384.000,-83.164,-176.100,9.315,148.764
C06109=1162.422,383.752,-83.129,-176.101,9.311,148.763
C06110=1162.426,383.505,-83.092,-176.102,9.308,148.762
C06111=1162.430,383.258,-83.056,-176.102,9.304,148.761
C06112=1162.435,383.010,-83.020,-176.103,9.301,148.761
C06113=1162.438,382.763,-82.984,-176.104,9.297,148.760
C06114=1162.442,382.515,-82.948,-176.105,9.294,148.759
C06115=1162.446,382.268,-82.912,-176.105,9.290,148.758
C06116=1162.449,382.021,-82.876,-176.107,9.286,148.758
C06117=1162.454,381.773,-82.840,-176.107,9.283,148.757
C06118=1162.458,381.526,-82.805,-176.108,9.280,148.756
C06119=1162.461,381.279,-82.768,-176.109,9.276,148.756
C06120=1162.466,381.031,-82.732,-176.110,9.273,148.755
C06121=1162.469,380.784,-82.697,-176.111,9.268,148.754
C06122=1162.473,380.536,-82.661,-176.112,9.265,148.754
C06123=1162.477,380.289,-82.624,-176.113,9.261,148.753
C06124=1162.481,380.042,-82.589,-176.114,9.257,148.752
C06125=1162.484,379.794,-82.553,-176.115,9.254,148.752
C06126=1162.489,379.546,-82.517,-176.116,9.250,148.751
C06127=1162.493,379.300,-82.481,-176.117,9.246,148.750
C06128=1162.496,379.053,-82.446,-176.118,9.243,148.750
C06129=1162.501,378.805,-82.410,-176.120,9.239,148.749
C06130=1162.505,378.557,-82.374,-176.121,9.235,148.748
C06131=1162.508,378.310,-82.338,-176.122,9.231,148.747
C06132=1162.513,378.062,-82.302,-176.123,9.228,148.747
C06133=1162.516,377.815,-82.266,-176.124,9.224,148.746
C06134=1162.520,377.568,-82.230,-176.126,9.220,148.746
C06135=1162.524,377.321,-82.195,-176.127,9.216,148.745
C06136=1162.528,377.073,-82.159,-176.129,9.212,148.744
C06137=1162.532,376.826,-82.124,-176.130,9.208,148.744
C06138=1162.536,376.578,-82.088,-176.132,9.204,148.743
C06139=1162.539,376.331,-82.053,-176.133,9.201,148.743
C06140=1162.544,376.083,-82.016,-176.134,9.197,148.742
C06141=1162.548,375.836,-81.981,-176.136,9.194,148.742
C06142=1162.552,375.588,-81.946,-176.137,9.190,148.741
C06143=1162.555,375.341,-81.910,-176.139,9.186,148.740
C06144=1162.559,375.094,-81.873,-176.140,9.182,148.740
C06145=1162.563,374.846,-81.838,-176.143,9.178,148.739
C06146=1162.567,374.599,-81.802,-176.144,9.174,148.739
C06147=1162.571,374.352,-81.767,-176.145,9.170,148.738
C06148=1162.575,374.104,-81.732,-176.147,9.166,148.738
C06149=1162.579,373.856,-81.697,-176.149,9.162,148.737
C06150=1162.583,373.609,-81.660,-176.151,9.159,148.736
C06151=1162.587,373.361,-81.625,-176.152,9.155,148.736
C06152=1162.591,373.114,-81.590,-176.154,9.151,148.735
C06153=1162.595,372.867,-81.554,-176.155,9.147,148.735
C06154=1162.598,372.619,-81.519,-176.158,9.143,148.734
C06155=1162.602,372.372,-81.483,-176.160,9.139,148.734
C06156=1162.606,372.125,-81.448,-176.161,9.136,148.733
C06157=1162.610,371.877,-81.412,-176.163,9.132,148.733
C06158=1162.614,371.630,-81.376,-176.165,9.128,148.732
C06159=1162.618,371.381,-81.341,-176.167,9.124,148.732
C06160=1162.622,371.135,-81.306,-176.169,9.120,148.731
C06161=1162.626,370.887,-81.271,-176.171,9.116,148.731
C06162=1162.630,370.640,-81.235,-176.173,9.112,148.730
C06163=1162.633,370.392,-81.200,-176.175,9.108,148.730
C06164=1162.638,370.145,-81.165,-176.177,9.105,148.730
C06165=1162.642,369.897,-81.130,-176.179,9.101,148.729
C06166=1162.645,369.650,-81.094,-176.181,9.096,148.728
C06167=1162.650,369.403,-81.059,-176.182,9.093,148.728
C06168=1162.654,369.155,-81.024,-176.184,9.089,148.728
C06169=1162.657,368.907,-80.988,-176.187,9.085,148.727
C06170=1162.661,368.660,-80.953,-176.189,9.082,148.727
C06171=1162.665,368.412,-80.918,-176.191,9.078,148.726
C06172=1162.669,368.165,-80.883,-176.193,9.074,148.726
C06173=1162.673,367.917,-80.847,-176.195,9.070,148.726
C06174=1162.677,367.670,-80.813,-176.198,9.066,148.725
C06175=1162.681,367.423,-80.777,-176.200,9.062,148.725
C06176=1162.685,367.175,-80.742,-176.201,9.058,148.724
C06177=1162.689,366.928,-80.707,-176.204,9.054,148.724
C06178=1162.693,366.680,-80.672,-176.206,9.051,148.724
C06179=1162.697,366.432,-80.637,-176.209,9.046,148.723
C06180=1162.701,366.185,-80.602,-176.211,9.043,148.723
C06181=1162.705,365.903,-80.562,-176.213,9.038,148.722
C06182=1162.710,365.620,-80.522,-176.216,9.034,148.722
C06183=1162.715,365.338,-80.482,-176.218,9.030,148.721
C06184=1162.719,365.055,-80.443,-176.221,9.025,148.721
C06185=1162.723,364.807,-80.407,-176.224,9.021,148.721
C06186=1162.727,364.559,-80.372,-176.225,9.018,148.720
C06187=1162.730,364.313,-80.338,-176.228,9.013,148.720
C06188=1162.734,364.065,-80.303,-176.230,9.010,148.720
C06189=1162.739,363.818,-80.268,-176.233,9.005,148.719
C06190=1162.743,363.570,-80.233,-176.235,9.002,148.719
C06191=1162.746,363.322,-80.197,-176.237,8.998,148.718
C06192=1162.750,363.075,-80.163,-176.240,8.994,148.718
C06193=1162.754,362.827,-80.128,-176.242,8.990,148.718
C06194=1162.758,362.580,-80.093,-176.244,8.987,148.717
C06195=1162.762,362.332,-80.058,-176.247,8.982,148.717
C06196=1162.767,362.085,-80.024,-176.249,8.979,148.717
C06197=1162.770,361.837,-79.989,-176.251,8.975,148.716
C06198=1162.774,361.589,-79.954,-176.254,8.971,148.716
C06199=1162.778,361.342,-79.920,-176.256,8.968,148.716
C06200=1162.782,361.094,-79.886,-176.259,8.964,148.715
C06201=1162.786,360.847,-79.850,-176.261,8.960,148.715
C06202=1162.790,360.599,-79.816,-176.263,8.956,148.715
C06203=1162.794,360.352,-79.781,-176.266,8.953,148.714
C06204=1162.798,360.104,-79.747,-176.268,8.948,148.714
C06205=1162.802,359.857,-79.712,-176.270,8.945,148.714
C06206=1162.806,359.609,-79.677,-176.273,8.941,148.714
C06207=1162.810,359.362,-79.643,-176.275,8.937,148.713
C06208=1162.814,359.114,-79.608,-176.278,8.933,148.713
C06209=1162.818,358.866,-79.574,-176.280,8.930,148.713
C06210=1162.821,358.619,-79.539,-176.283,8.925,148.712
C06211=1162.826,358.371,-79.505,-176.285,8.922,148.712
C06212=1162.830,358.123,-79.470,-176.287,8.919,148.712
C06213=1162.834,357.876,-79.436,-176.290,8.915,148.711
C06214=1162.838,357.628,-79.401,-176.292,8.911,148.711
C06215=1162.841,357.381,-79.367,-176.295,8.907,148.711
C06216=1162.845,357.133,-79.332,-176.297,8.904,148.711
C06217=1162.850,356.886,-79.298,-176.300,8.899,148.710
C06218=1162.854,356.639,-79.264,-176.302,8.896,148.710
C06219=1162.858,356.391,-79.229,-176.304,8.893,148.710
C06220=1162.862,356.143,-79.195,-176.307,8.888,148.709
C06221=1162.866,355.895,-79.160,-176.309,8.885,148.709
C06222=1162.870,355.648,-79.127,-176.312,8.881,148.709
C06223=1162.874,355.399,-79.092,-176.314,8.878,148.708
C06224=1162.877,355.152,-79.058,-176.316,8.874,148.708
C06225=1162.882,354.905,-79.024,-176.319,8.870,148.708
C06226=1162.885,354.657,-78.990,-176.321,8.867,148.708
C06227=1162.890,354.410,-78.955,-176.324,8.862,148.707
C06228=1162.893,354.162,-78.921,-176.326,8.859,148.707
C06229=1162.898,353.914,-78.886,-176.328,8.856,148.707
C06230=1162.901,353.667,-78.852,-176.331,8.851,148.706
C06231=1162.906,353.419,-78.818,-176.334,8.848,148.706
C06232=1162.910,353.171,-78.785,-176.336,8.844,148.706
C06233=1162.914,352.924,-78.750,-176.338,8.840,148.706
C06234=1162.917,352.676,-78.716,-176.341,8.837,148.705
C06235=1162.922,352.428,-78.682,-176.343,8.833,148.705
C06236=1162.926,352.181,-78.648,-176.346,8.830,148.705
C06237=1162.929,351.933,-78.614,-176.349,8.826,148.705
C06238=1162.934,351.686,-78.579,-176.350,8.822,148.704
C06239=1162.938,351.438,-78.546,-176.353,8.819,148.704
C06240=1162.942,351.190,-78.511,-176.356,8.815,148.704
C06241=1162.946,350.943,-78.478,-176.358,8.811,148.703
C06242=1162.950,350.695,-78.444,-176.360,8.808,148.703
C06243=1162.954,350.447,-78.410,-176.363,8.804,148.703
C06244=1162.958,350.200,-78.376,-176.365,8.800,148.703
C06245=1162.962,349.952,-78.343,-176.367,8.797,148.702
C06246=1162.966,349.704,-78.308,-176.370,8.793,148.702
C06247=1162.970,349.456,-78.275,-176.372,8.790,148.702
C06248=1162.974,349.209,-78.241,-176.375,8.786,148.702
C06249=1162.978,348.962,-78.206,-176.378,8.782,148.701
C06250=1162.982,348.713,-78.173,-176.380,8.779,148.701
C06251=1162.986,348.466,-78.139,-176.383,8.775,148.701
C06252=1162.991,348.218,-78.105,-176.385,8.771,148.701
C06253=1162.994,347.971,-78.071,-176.387,8.768,148.700
C06254=1162.998,347.723,-78.038,-176.390,8.764,148.700
C06255=1163.002,347.476,-78.004,-176.392,8.761,148.700
C06256=1163.007,347.228,-77.970,-176.394,8.757,148.700
C06257=1163.011,346.980,-77.936,-176.397,8.753,148.699
C06258=1163.014,346.732,-77.903,-176.400,8.750,148.699
C06259=1163.018,346.484,-77.870,-176.402,8.747,148.699
C06260=1163.023,346.237,-77.835,-176.405,8.743,148.699
C06261=1163.027,345.989,-77.802,-176.407,8.739,148.698
C06262=1163.031,345.742,-77.768,-176.409,8.736,148.698
C06263=1163.034,345.494,-77.735,-176.412,8.732,148.698
C06264=1163.038,345.246,-77.701,-176.415,8.729,148.698
C06265=1163.043,344.998,-77.667,-176.416,8.725,148.697
C06266=1163.047,344.751,-77.634,-176.419,8.721,148.697
C06267=1163.051,344.503,-77.601,-176.422,8.718,148.697
C06268=1163.055,344.256,-77.567,-176.424,8.714,148.697
C06269=1163.059,344.007,-77.533,-176.427,8.710,148.696
C06270=1163.063,343.760,-77.500,-176.429,8.707,148.696
C06271=1163.068,343.512,-77.466,-176.431,8.704,148.696
C06272=1163.071,343.265,-77.432,-176.434,8.699,148.696
C06273=1163.076,343.017,-77.399,-176.437,8.696,148.696
C06274=1163.080,342.769,-77.366,-176.439,8.693,148.695
C06275=1163.084,342.521,-77.333,-176.442,8.689,148.695
C06276=1163.087,342.273,-77.299,-176.444,8.685,148.695
C06277=1163.092,342.025,-77.266,-176.446,8.682,148.695
C06278=1163.095,341.778,-77.232,-176.449,8.679,148.694
C06279=1163.100,341.530,-77.199,-176.451,8.675,148.694
C06280=1163.104,341.283,-77.166,-176.454,8.671,148.694
C06281=1163.108,341.035,-77.133,-176.456,8.668,148.694
C06282=1163.112,340.787,-77.100,-176.459,8.664,148.694
C06283=1163.116,340.540,-77.067,-176.461,8.661,148.693
C06284=1163.120,340.292,-77.033,-176.464,8.657,148.693
C06285=1163.125,340.012,-76.996,-176.466,8.653,148.693
C06286=1163.130,339.732,-76.958,-176.470,8.650,148.693
C06287=1163.134,339.453,-76.921,-176.473,8.645,148.693
C06288=1163.139,339.173,-76.883,-176.475,8.641,148.692
C06289=1163.143,338.926,-76.850,-176.478,8.638,148.692
C06290=1163.147,338.678,-76.817,-176.480,8.635,148.692
C06291=1163.151,338.430,-76.784,-176.482,8.631,148.692
C06292=1163.155,338.182,-76.750,-176.485,8.627,148.691
C06293=1163.159,337.934,-76.717,-176.488,8.624,148.691
C06294=1163.163,337.686,-76.684,-176.490,8.621,148.691
C06295=1163.167,337.439,-76.651,-176.492,8.618,148.691
C06296=1163.171,337.190,-76.618,-176.495,8.613,148.691
C06297=1163.176,336.943,-76.585,-176.497,8.610,148.690
C06298=1163.180,336.695,-76.552,-176.500,8.607,148.690
C06299=1163.183,336.447,-76.520,-176.503,8.603,148.690
C06300=1163.187,336.200,-76.486,-176.505,8.600,148.690
C06301=1163.191,335.952,-76.453,-176.507,8.596,148.690
C06302=1163.196,335.704,-76.421,-176.510,8.593,148.690
C06303=1163.200,335.456,-76.388,-176.513,8.589,148.689
C06304=1163.204,335.208,-76.355,-176.515,8.586,148.689
C06305=1163.208,334.961,-76.322,-176.517,8.582,148.689
C06306=1163.212,334.713,-76.289,-176.520,8.579,148.689
C06307=1163.216,334.465,-76.256,-176.523,8.575,148.689
C06308=1163.220,334.217,-76.223,-176.525,8.572,148.688
C06309=1163.224,333.969,-76.190,-176.527,8.569,148.688
C06310=1163.229,333.722,-76.159,-176.530,8.566,148.688
C06311=1163.233,333.474,-76.125,-176.533,8.561,148.688
C06312=1163.237,333.226,-76.092,-176.535,8.558,148.688
C06313=1163.241,332.978,-76.060,-176.537,8.555,148.687
C06314=1163.245,332.731,-76.027,-176.540,8.552,148.687
C06315=1163.249,332.483,-75.994,-176.543,8.548,148.687
C06316=1163.253,332.235,-75.962,-176.545,8.544,148.687
C06317=1163.258,331.987,-75.929,-176.547,8.541,148.687
C06318=1163.261,331.739,-75.896,-176.550,8.538,148.686
C06319=1163.265,331.491,-75.864,-176.553,8.534,148.686
C06320=1163.270,331.243,-75.830,-176.555,8.531,148.686
C06321=1163.273,330.995,-75.799,-176.558,8.528,148.686
C06322=1163.278,330.748,-75.766,-176.560,8.524,148.686
C06323=1163.282,330.500,-75.733,-176.562,8.521,148.686
C06324=1163.286,330.252,-75.701,-176.565,8.517,148.685
C06325=1163.290,330.004,-75.668,-176.568,8.514,148.685
C06326=1163.294,329.756,-75.635,-176.570,8.511,148.685
C06327=1163.298,329.508,-75.603,-176.572,8.507,148.685
C06328=1163.302,329.261,-75.570,-176.575,8.503,148.685
C06329=1163.307,329.013,-75.539,-176.578,8.500,148.685
C06330=1163.311,328.765,-75.506,-176.580,8.497,148.685
C06331=1163.315,328.517,-75.473,-176.583,8.494,148.684
C06332=1163.319,328.269,-75.441,-176.585,8.490,148.684
C06333=1163.323,328.021,-75.408,-176.588,8.486,148.684
C06334=1163.327,327.773,-75.376,-176.591,8.483,148.684
C06335=1163.332,327.526,-75.344,-176.593,8.480,148.684
C06336=1163.335,327.278,-75.312,-176.595,8.477,148.684
C06337=1163.340,327.030,-75.279,-176.597,8.473,148.683
C06338=1163.344,326.782,-75.247,-176.601,8.470,148.683
C06339=1163.347,326.534,-75.214,-176.603,8.466,148.683
C06340=1163.352,326.287,-75.182,-176.605,8.463,148.683
C06341=1163.356,326.039,-75.150,-176.608,8.460,148.683
C06342=1163.361,325.790,-75.118,-176.610,8.457,148.683
C06343=1163.364,325.543,-75.085,-176.613,8.453,148.682
C06344=1163.368,325.295,-75.053,-176.616,8.449,148.682
C06345=1163.373,325.047,-75.021,-176.618,8.446,148.682
C06346=1163.376,324.799,-74.989,-176.621,8.443,148.682
C06347=1163.381,324.551,-74.956,-176.623,8.440,148.682
C06348=1163.384,324.303,-74.924,-176.626,8.436,148.682
C06349=1163.389,324.056,-74.892,-176.629,8.433,148.682
C06350=1163.393,323.808,-74.861,-176.631,8.429,148.681
C06351=1163.397,323.559,-74.828,-176.633,8.426,148.681
C06352=1163.401,323.311,-74.796,-176.635,8.423,148.681
C06353=1163.405,323.064,-74.765,-176.639,8.419,148.681
C06354=1163.410,322.816,-74.732,-176.641,8.416,148.681
C06355=1163.413,322.568,-74.700,-176.643,8.412,148.681
C06356=1163.418,322.321,-74.668,-176.646,8.409,148.681
C06357=1163.422,322.072,-74.636,-176.648,8.406,148.680
C06358=1163.426,321.824,-74.604,-176.651,8.403,148.680
C06359=1163.430,321.576,-74.572,-176.654,8.399,148.680
C06360=1163.435,321.329,-74.540,-176.656,8.396,148.680
C06361=1163.438,321.081,-74.508,-176.659,8.393,148.680
C06362=1163.442,320.833,-74.476,-176.661,8.390,148.680
C06363=1163.447,320.585,-74.444,-176.664,8.386,148.680
C06364=1163.451,320.337,-74.412,-176.666,8.383,148.679
C06365=1163.454,320.089,-74.381,-176.669,8.379,148.679
C06366=1163.460,319.841,-74.349,-176.672,8.376,148.679
C06367=1163.463,319.593,-74.317,-176.674,8.373,148.679
C06368=1163.467,319.345,-74.286,-176.677,8.370,148.679
C06369=1163.471,319.097,-74.254,-176.679,8.366,148.679
C06370=1163.476,318.849,-74.222,-176.681,8.363,148.679
C06371=1163.480,318.602,-74.190,-176.684,8.359,148.679
C06372=1163.484,318.353,-74.158,-176.687,8.356,148.678
C06373=1163.488,318.105,-74.126,-176.689,8.353,148.678
C06374=1163.492,317.857,-74.096,-176.692,8.350,148.678
C06375=1163.497,317.609,-74.063,-176.694,8.346,148.678
C06376=1163.500,317.361,-74.031,-176.697,8.343,148.678
C06377=1163.505,317.114,-74.000,-176.699,8.340,148.678
C06378=1163.509,316.865,-73.969,-176.702,8.336,148.678
C06379=1163.513,316.618,-73.937,-176.705,8.333,148.678
C06380=1163.517,316.369,-73.905,-176.707,8.330,148.677
C06381=1163.521,316.121,-73.873,-176.709,8.327,148.677
C06382=1163.526,315.873,-73.842,-176.712,8.324,148.677
C06383=1163.530,315.625,-73.810,-176.714,8.320,148.677
C06384=1163.534,315.378,-73.779,-176.717,8.317,148.677
C06385=1163.538,315.129,-73.748,-176.720,8.313,148.677
C06386=1163.542,314.882,-73.716,-176.722,8.310,148.677
C06387=1163.546,314.634,-73.685,-176.725,8.307,148.677
C06388=1163.550,314.386,-73.654,-176.727,8.304,148.677
C06389=1163.555,314.109,-73.618,-176.731,8.300,148.677
C06390=1163.560,313.832,-73.583,-176.733,8.297,148.676
C06391=1163.565,313.555,-73.548,-176.736,8.293,148.676
C06392=1163.569,313.277,-73.513,-176.739,8.289,148.676
C06393=1163.574,313.029,-73.481,-176.742,8.286,148.676
C06394=1163.578,312.781,-73.450,-176.744,8.282,148.676
C06395=1163.582,312.533,-73.419,-176.746,8.279,148.676
C06396=1163.586,312.285,-73.388,-176.749,8.276,148.676
C06397=1163.590,312.037,-73.356,-176.752,8.273,148.676
C06398=1163.594,311.789,-73.325,-176.754,8.270,148.676
C06399=1163.599,311.541,-73.293,-176.757,8.267,148.675
C06400=1163.603,311.293,-73.262,-176.759,8.264,148.675
C06401=1163.607,311.045,-73.231,-176.762,8.259,148.675
C06402=1163.611,310.797,-73.200,-176.765,8.257,148.675
C06403=1163.615,310.549,-73.168,-176.767,8.253,148.675
C06404=1163.620,310.301,-73.137,-176.770,8.250,148.675
C06405=1163.624,310.053,-73.106,-176.772,8.247,148.675
C06406=1163.628,309.805,-73.075,-176.775,8.244,148.675
C06407=1163.632,309.557,-73.044,-176.777,8.241,148.675
C06408=1163.637,309.309,-73.013,-176.780,8.237,148.674
C06409=1163.640,309.061,-72.982,-176.782,8.234,148.674
C06410=1163.644,308.813,-72.951,-176.785,8.231,148.674
C06411=1163.649,308.565,-72.920,-176.788,8.227,148.674
C06412=1163.653,308.317,-72.888,-176.790,8.224,148.674
C06413=1163.657,308.069,-72.858,-176.793,8.221,148.674
C06414=1163.661,307.821,-72.826,-176.795,8.218,148.674
C06415=1163.666,307.573,-72.796,-176.798,8.215,148.674
C06416=1163.670,307.325,-72.764,-176.800,8.212,148.674
C06417=1163.673,307.077,-72.734,-176.803,8.209,148.674
C06418=1163.678,306.829,-72.703,-176.805,8.205,148.674
C06419=1163.682,306.580,-72.672,-176.808,8.202,148.674
C06420=1163.687,306.332,-72.641,-176.810,8.199,148.673
C06421=1163.691,306.085,-72.610,-176.813,8.196,148.673
C06422=1163.695,305.836,-72.578,-176.816,8.192,148.673
C06423=1163.699,305.589,-72.548,-176.819,8.189,148.673
C06424=1163.703,305.341,-72.517,-176.821,8.186,148.673
C06425=1163.707,305.092,-72.486,-176.824,8.183,148.673
C06426=1163.712,304.844,-72.456,-176.827,8.180,148.673
C06427=1163.716,304.596,-72.425,-176.829,8.176,148.673
C06428=1163.720,304.348,-72.394,-176.832,8.174,148.673
C06429=1163.725,304.100,-72.364,-176.834,8.170,148.673
C06430=1163.729,303.852,-72.333,-176.837,8.167,148.673
C06431=1163.732,303.604,-72.302,-176.839,8.164,148.673
C06432=1163.737,303.356,-72.271,-176.842,8.161,148.673
C06433=1163.742,303.108,-72.241,-176.844,8.158,148.672
C06434=1163.746,302.860,-72.210,-176.847,8.155,148.672
C06435=1163.750,302.611,-72.179,-176.850,8.151,148.672
C06436=1163.754,302.363,-72.149,-176.852,8.148,148.672
C06437=1163.759,302.115,-72.118,-176.855,8.145,148.672
C06438=1163.763,301.868,-72.088,-176.857,8.141,148.672
C06439=1163.767,301.619,-72.057,-176.860,8.138,148.672
C06440=1163.771,301.371,-72.026,-176.862,8.135,148.672
C06441=1163.775,301.123,-71.996,-176.865,8.132,148.672
C06442=1163.780,300.876,-71.965,-176.868,8.129,148.672
C06443=1163.783,300.627,-71.934,-176.870,8.126,148.672
C06444=1163.788,300.379,-71.904,-176.873,8.123,148.672
C06445=1163.793,300.131,-71.874,-176.875,8.120,148.672
C06446=1163.796,299.883,-71.843,-176.878,8.117,148.672
C06447=1163.801,299.634,-71.812,-176.880,8.113,148.672
C06448=1163.804,299.387,-71.782,-176.883,8.110,148.672
C06449=1163.809,299.139,-71.751,-176.885,8.107,148.671
C06450=1163.814,298.890,-71.721,-176.888,8.104,148.671
C06451=1163.817,298.642,-71.691,-176.891,8.101,148.671
C06452=1163.822,298.394,-71.660,-176.893,8.098,148.671
C06453=1163.826,298.146,-71.630,-176.897,8.094,148.671
C06454=1163.831,297.898,-71.600,-176.899,8.091,148.671
C06455=1163.834,297.650,-71.570,-176.902,8.088,148.671
C06456=1163.839,297.402,-71.539,-176.904,8.085,148.671
C06457=1163.843,297.153,-71.509,-176.907,8.082,148.671
C06458=1163.847,296.905,-71.478,-176.909,8.079,148.671
C06459=1163.851,296.657,-71.448,-176.912,8.076,148.671
C06460=1163.856,296.409,-71.418,-176.914,8.072,148.671
C06461=1163.860,296.161,-71.388,-176.917,8.069,148.671
C06462=1163.864,295.913,-71.358,-176.919,8.066,148.671
C06463=1163.868,295.664,-71.327,-176.922,8.063,148.671
C06464=1163.872,295.417,-71.297,-176.925,8.060,148.671
C06465=1163.877,295.168,-71.267,-176.927,8.057,148.671
C06466=1163.881,294.920,-71.237,-176.930,8.054,148.671
C06467=1163.886,294.672,-71.207,-176.933,8.051,148.671
C06468=1163.890,294.424,-71.177,-176.935,8.048,148.670
C06469=1163.894,294.176,-71.147,-176.938,8.045,148.670
C06470=1163.898,293.928,-71.116,-176.941,8.042,148.670
C06471=1163.902,293.679,-71.087,-176.943,8.039,148.670
C06472=1163.906,293.431,-71.056,-176.946,8.036,148.670
C06473=1163.911,293.183,-71.026,-176.948,8.033,148.670
C06474=1163.915,292.935,-70.996,-176.951,8.029,148.670
C06475=1163.919,292.687,-70.967,-176.953,8.026,148.670
C06476=1163.923,292.439,-70.936,-176.956,8.023,148.670
C06477=1163.928,292.191,-70.907,-176.958,8.020,148.670
C06478=1163.932,291.942,-70.877,-176.961,8.017,148.670
C06479=1163.936,291.694,-70.846,-176.964,8.014,148.670
C06480=1163.941,291.446,-70.817,-176.966,8.011,148.670
C06481=1163.945,291.198,-70.787,-176.969,8.008,148.670
C06482=1163.949,290.950,-70.757,-176.972,8.005,148.670
C06483=1163.954,290.702,-70.727,-176.974,8.002,148.670
C06484=1163.958,290.453,-70.698,-176.977,7.999,148.670
C06485=1163.962,290.206,-70.668,-176.980,7.996,148.670
C06486=1163.967,289.957,-70.638,-176.982,7.993,148.670
C06487=1163.971,289.709,-70.608,-176.985,7.989,148.670
C06488=1163.975,289.461,-70.579,-176.987,7.987,148.670
C06489=1163.978,289.212,-70.548,-176.990,7.984,148.670
C06490=1163.982,288.964,-70.519,-176.992,7.980,148.670
C06491=1163.988,288.716,-70.489,-176.995,7.977,148.670
C06492=1163.992,288.468,-70.460,-176.998,7.974,148.670
C06493=1163.997,288.193,-70.426,-177.001,7.971,148.670
C06494=1164.002,287.918,-70.394,-177.003,7.967,148.670
C06495=1164.006,287.643,-70.361,-177.006,7.964,148.670
C06496=1164.011,287.368,-70.328,-177.010,7.961,148.670
C06497=1164.014,287.120,-70.298,-177.012,7.958,148.670
C06498=1164.019,286.872,-70.268,-177.015,7.954,148.669
C06499=1164.023,286.623,-70.239,-177.017,7.951,148.670
C06500=1164.028,286.375,-70.209,-177.020,7.948,148.670
C06501=1164.032,286.127,-70.180,-177.023,7.945,148.670
C06502=1164.036,285.879,-70.150,-177.025,7.942,148.669
C06503=1164.040,285.630,-70.121,-177.028,7.939,148.669
C06504=1164.044,285.382,-70.091,-177.031,7.936,148.670
C06505=1164.049,285.134,-70.062,-177.033,7.933,148.670
C06506=1164.053,284.886,-70.032,-177.036,7.930,148.669
C06507=1164.058,284.638,-70.003,-177.038,7.927,148.669
C06508=1164.062,284.390,-69.974,-177.041,7.925,148.670
C06509=1164.067,284.141,-69.944,-177.043,7.922,148.670
C06510=1164.071,283.893,-69.914,-177.046,7.919,148.669
C06511=1164.075,283.645,-69.885,-177.048,7.916,148.669
C06512=1164.079,283.396,-69.855,-177.051,7.913,148.669
C06513=1164.083,283.148,-69.826,-177.054,7.910,148.669
C06514=1164.088,282.900,-69.797,-177.057,7.907,148.670
C06515=1164.092,282.651,-69.767,-177.059,7.903,148.669
C06516=1164.097,282.403,-69.739,-177.062,7.900,148.669
C06517=1164.101,282.155,-69.709,-177.065,7.897,148.669
C06518=1164.105,281.907,-69.680,-177.067,7.895,148.669
C06519=1164.109,281.659,-69.650,-177.070,7.891,148.669
C06520=1164.113,281.411,-69.622,-177.072,7.888,148.669
C06521=1164.117,281.162,-69.592,-177.075,7.885,148.669
C06522=1164.122,280.914,-69.564,-177.078,7.882,148.669
C06523=1164.126,280.666,-69.534,-177.081,7.879,148.669
C06524=1164.130,280.418,-69.505,-177.083,7.876,148.669
C06525=1164.135,280.169,-69.475,-177.086,7.873,148.669
C06526=1164.139,279.920,-69.447,-177.088,7.870,148.669
C06527=1164.144,279.673,-69.418,-177.091,7.867,148.669
C06528=1164.148,279.425,-69.388,-177.094,7.864,148.669
C06529=1164.152,279.176,-69.359,-177.096,7.862,148.670
C06530=1164.156,278.928,-69.330,-177.098,7.859,148.669
C06531=1164.160,278.679,-69.301,-177.101,7.856,148.669
C06532=1164.165,278.432,-69.272,-177.104,7.853,148.669
C06533=1164.169,278.183,-69.243,-177.107,7.850,148.670
C06534=1164.174,277.935,-69.214,-177.109,7.847,148.670
C06535=1164.178,277.686,-69.185,-177.112,7.844,148.670
C06536=1164.182,277.438,-69.156,-177.114,7.841,148.669
C06537=1164.186,277.190,-69.127,-177.117,7.838,148.669
C06538=1164.191,276.941,-69.098,-177.120,7.835,148.670
C06539=1164.195,276.693,-69.069,-177.123,7.832,148.670
C06540=1164.199,276.445,-69.041,-177.125,7.829,148.670
C06541=1164.204,276.197,-69.012,-177.128,7.826,148.670
C06542=1164.208,275.948,-68.983,-177.130,7.823,148.670
C06543=1164.212,275.700,-68.953,-177.133,7.821,148.670
C06544=1164.217,275.452,-68.926,-177.135,7.818,148.670
C06545=1164.221,275.204,-68.896,-177.138,7.815,148.670
C06546=1164.225,274.955,-68.867,-177.141,7.812,148.670
C06547=1164.229,274.707,-68.838,-177.144,7.809,148.670
C06548=1164.234,274.459,-68.810,-177.146,7.806,148.670
C06549=1164.238,274.210,-68.781,-177.149,7.803,148.670
C06550=1164.242,273.962,-68.752,-177.151,7.799,148.670
C06551=1164.246,273.714,-68.724,-177.154,7.797,148.670
C06552=1164.251,273.465,-68.695,-177.157,7.794,148.670
C06553=1164.255,273.217,-68.666,-177.160,7.791,148.670
C06554=1164.260,272.969,-68.638,-177.162,7.788,148.670
C06555=1164.264,272.720,-68.609,-177.165,7.785,148.670
C06556=1164.268,272.471,-68.580,-177.167,7.783,148.670
C06557=1164.273,272.224,-68.552,-177.170,7.780,148.670
C06558=1164.277,271.975,-68.523,-177.173,7.777,148.670
C06559=1164.282,271.726,-68.494,-177.175,7.773,148.670
C06560=1164.286,271.479,-68.466,-177.178,7.770,148.670
C06561=1164.290,271.230,-68.437,-177.181,7.767,148.670
C06562=1164.294,270.982,-68.409,-177.184,7.764,148.670
C06563=1164.299,270.734,-68.380,-177.186,7.762,148.670
C06564=1164.302,270.486,-68.352,-177.188,7.759,148.670
C06565=1164.307,270.237,-68.323,-177.191,7.756,148.670
C06566=1164.312,269.989,-68.294,-177.194,7.753,148.670
C06567=1164.316,269.741,-68.267,-177.197,7.750,148.670
C06568=1164.320,269.492,-68.237,-177.199,7.748,148.670
C06569=1164.324,269.244,-68.209,-177.202,7.745,148.671
C06570=1164.329,268.996,-68.181,-177.205,7.742,148.671
C06571=1164.333,268.747,-68.153,-177.207,7.739,148.670
C06572=1164.338,268.499,-68.124,-177.209,7.736,148.670
C06573=1164.342,268.250,-68.096,-177.212,7.733,148.671
C06574=1164.347,268.002,-68.068,-177.215,7.730,148.671
C06575=1164.351,267.754,-68.040,-177.218,7.727,148.671
C06576=1164.355,267.505,-68.010,-177.221,7.724,148.671
C06577=1164.359,267.257,-67.982,-177.223,7.721,148.671
C06578=1164.364,267.008,-67.954,-177.226,7.718,148.671
C06579=1164.368,266.761,-67.926,-177.228,7.716,148.671
C06580=1164.372,266.512,-67.898,-177.231,7.713,148.671
C06581=1164.377,266.264,-67.869,-177.234,7.710,148.671
C06582=1164.381,266.015,-67.841,-177.236,7.707,148.671
C06583=1164.386,265.767,-67.813,-177.239,7.704,148.671
C06584=1164.389,265.519,-67.785,-177.242,7.702,148.671
C06585=1164.395,265.270,-67.756,-177.245,7.699,148.671
C06586=1164.398,265.022,-67.728,-177.247,7.696,148.671
C06587=1164.403,264.774,-67.700,-177.250,7.693,148.671
C06588=1164.407,264.524,-67.672,-177.252,7.690,148.671
C06589=1164.412,264.276,-67.645,-177.255,7.688,148.671
C06590=1164.416,264.028,-67.616,-177.258,7.685,148.672
C06591=1164.421,263.780,-67.588,-177.261,7.682,148.672
C06592=1164.425,263.532,-67.560,-177.263,7.679,148.672
C06593=1164.429,263.283,-67.532,-177.266,7.677,148.672
C06594=1164.434,263.035,-67.504,-177.268,7.674,148.672
C06595=1164.438,262.786,-67.476,-177.271,7.671,148.672
C06596=1164.442,262.538,-67.448,-177.274,7.668,148.672
C06597=1164.447,262.265,-67.418,-177.277,7.665,148.672
C06598=1164.451,261.992,-67.386,-177.279,7.662,148.672
C06599=1164.457,261.718,-67.355,-177.283,7.658,148.672
C06600=1164.461,261.445,-67.324,-177.286,7.655,148.672
C06601=1164.466,261.196,-67.297,-177.288,7.652,148.672
C06602=1164.470,260.949,-67.270,-177.290,7.650,148.672
C06603=1164.474,260.700,-67.241,-177.293,7.647,148.672
C06604=1164.478,260.452,-67.214,-177.296,7.644,148.672
C06605=1164.483,260.203,-67.186,-177.299,7.641,148.672
C06606=1164.488,259.955,-67.158,-177.302,7.638,148.672
C06607=1164.492,259.707,-67.130,-177.304,7.635,148.673
C06608=1164.496,259.458,-67.103,-177.306,7.633,148.673
C06609=1164.500,259.210,-67.075,-177.309,7.630,148.673
C06610=1164.505,258.961,-67.046,-177.312,7.627,148.673
C06611=1164.509,258.712,-67.019,-177.315,7.624,148.673
C06612=1164.514,258.465,-66.991,-177.318,7.622,148.673
C06613=1164.518,258.215,-66.964,-177.320,7.619,148.673
C06614=1164.522,257.968,-66.936,-177.323,7.616,148.673
C06615=1164.527,257.719,-66.909,-177.326,7.613,148.673
C06616=1164.531,257.470,-66.880,-177.328,7.611,148.673
C06617=1164.536,257.222,-66.853,-177.331,7.608,148.673
C06618=1164.540,256.974,-66.826,-177.333,7.605,148.673
C06619=1164.544,256.725,-66.797,-177.336,7.602,148.674
C06620=1164.549,256.477,-66.770,-177.339,7.600,148.674
C06621=1164.553,256.229,-66.743,-177.342,7.597,148.674
C06622=1164.557,255.980,-66.715,-177.344,7.594,148.674
C06623=1164.562,255.732,-66.687,-177.347,7.591,148.674
C06624=1164.566,255.483,-66.660,-177.349,7.589,148.674
C06625=1164.571,255.235,-66.633,-177.353,7.586,148.674
C06626=1164.575,254.986,-66.605,-177.355,7.583,148.674
C06627=1164.579,254.738,-66.578,-177.358,7.580,148.674
C06628=1164.584,254.490,-66.550,-177.360,7.578,148.674
C06629=1164.588,254.241,-66.523,-177.363,7.575,148.674
C06630=1164.592,253.992,-66.496,-177.366,7.572,148.674
C06631=1164.597,253.744,-66.468,-177.369,7.569,148.675
C06632=1164.601,253.496,-66.441,-177.371,7.567,148.675
C06633=1164.605,253.247,-66.413,-177.374,7.564,148.675
C06634=1164.610,252.999,-66.386,-177.376,7.561,148.675
C06635=1164.614,252.750,-66.359,-177.379,7.558,148.675
C06636=1164.619,252.502,-66.332,-177.382,7.555,148.675
C06637=1164.623,252.254,-66.304,-177.384,7.553,148.675
C06638=1164.627,252.005,-66.276,-177.387,7.550,148.675
C06639=1164.632,251.756,-66.249,-177.390,7.547,148.675
C06640=1164.637,251.508,-66.222,-177.393,7.544,148.675
C06641=1164.641,251.260,-66.194,-177.395,7.542,148.676
C06642=1164.645,251.011,-66.167,-177.398,7.539,148.676
C06643=1164.650,250.762,-66.140,-177.401,7.537,148.676
C06644=1164.654,250.514,-66.114,-177.404,7.534,148.676
C06645=1164.658,250.265,-66.086,-177.406,7.532,148.676
C06646=1164.663,250.017,-66.059,-177.409,7.529,148.676
C06647=1164.667,249.769,-66.032,-177.411,7.526,148.676
C06648=1164.672,249.520,-66.004,-177.414,7.523,148.676
C06649=1164.676,249.271,-65.977,-177.416,7.521,148.676
C06650=1164.681,249.023,-65.950,-177.420,7.518,148.677
C06651=1164.685,248.775,-65.924,-177.422,7.515,148.677
C06652=1164.689,248.526,-65.897,-177.425,7.512,148.677
C06653=1164.694,248.278,-65.869,-177.427,7.510,148.677
C06654=1164.698,248.028,-65.842,-177.430,7.507,148.677
C06655=1164.703,247.780,-65.815,-177.433,7.504,148.677
C06656=1164.707,247.532,-65.789,-177.436,7.501,148.677
C06657=1164.711,247.283,-65.761,-177.438,7.499,148.677
C06658=1164.716,247.035,-65.734,-177.441,7.496,148.677
C06659=1164.721,246.786,-65.707,-177.444,7.493,148.677
C06660=1164.725,246.538,-65.680,-177.446,7.490,148.678
C06661=1164.729,246.290,-65.654,-177.449,7.488,148.678
C06662=1164.734,246.041,-65.627,-177.452,7.486,148.678
C06663=1164.738,245.792,-65.599,-177.455,7.483,148.678
C06664=1164.742,245.544,-65.573,-177.457,7.480,148.678
C06665=1164.747,245.295,-65.546,-177.460,7.478,148.678
C06666=1164.751,245.047,-65.519,-177.462,7.475,148.678
C06667=1164.756,244.798,-65.492,-177.466,7.472,148.679
C06668=1164.760,244.550,-65.465,-177.468,7.470,148.679
C06669=1164.764,244.302,-65.438,-177.471,7.467,148.679
C06670=1164.769,244.052,-65.412,-177.473,7.464,148.679
C06671=1164.773,243.804,-65.385,-177.476,7.461,148.679
C06672=1164.778,243.556,-65.358,-177.479,7.459,148.679
C06673=1164.783,243.307,-65.331,-177.482,7.456,148.679
C06674=1164.787,243.059,-65.305,-177.484,7.453,148.679
C06675=1164.791,242.810,-65.278,-177.486,7.451,148.679
C06676=1164.795,242.562,-65.252,-177.490,7.449,148.680
C06677=1164.800,242.313,-65.225,-177.492,7.446,148.680
C06678=1164.805,242.065,-65.198,-177.495,7.444,148.680
C06679=1164.809,241.816,-65.172,-177.497,7.441,148.680
C06680=1164.814,241.567,-65.145,-177.500,7.438,148.680
C06681=1164.818,241.319,-65.119,-177.503,7.435,148.680
C06682=1164.822,241.071,-65.091,-177.506,7.433,148.680
C06683=1164.826,240.822,-65.066,-177.508,7.430,148.680
C06684=1164.831,240.573,-65.039,-177.511,7.427,148.681
C06685=1164.836,240.325,-65.012,-177.514,7.425,148.681
C06686=1164.840,240.076,-64.986,-177.517,7.422,148.681
C06687=1164.845,239.828,-64.959,-177.519,7.419,148.681
C06688=1164.849,239.580,-64.932,-177.521,7.417,148.681
C06689=1164.853,239.330,-64.906,-177.525,7.415,148.681
C06690=1164.857,239.082,-64.879,-177.527,7.412,148.681
C06691=1164.862,238.833,-64.853,-177.530,7.410,148.682
C06692=1164.866,238.585,-64.827,-177.533,7.407,148.682
C06693=1164.871,238.336,-64.800,-177.536,7.404,148.682
C06694=1164.875,238.088,-64.774,-177.538,7.402,148.682
C06695=1164.880,237.838,-64.748,-177.541,7.399,148.682
C06696=1164.884,237.590,-64.721,-177.544,7.396,148.682
C06697=1164.888,237.342,-64.695,-177.546,7.394,148.683
C06698=1164.894,237.094,-64.669,-177.549,7.391,148.683
C06699=1164.898,236.845,-64.643,-177.552,7.388,148.683
C06700=1164.902,236.596,-64.616,-177.554,7.386,148.683
C06701=1164.907,236.325,-64.587,-177.557,7.384,148.683
C06702=1164.912,236.053,-64.558,-177.560,7.381,148.683
C06703=1164.917,235.782,-64.530,-177.563,7.378,148.683
C06704=1164.921,235.510,-64.502,-177.566,7.375,148.684
C06705=1164.926,235.261,-64.475,-177.569,7.372,148.684
C06706=1164.930,235.012,-64.449,-177.572,7.369,148.684
C06707=1164.934,234.764,-64.423,-177.574,7.367,148.684
C06708=1164.939,234.515,-64.396,-177.577,7.365,148.684
C06709=1164.943,234.266,-64.370,-177.580,7.362,148.684
C06710=1164.949,234.018,-64.344,-177.582,7.360,148.684
C06711=1164.953,233.770,-64.318,-177.585,7.357,148.685
C06712=1164.957,233.521,-64.292,-177.588,7.354,148.685
C06713=1164.961,233.272,-64.266,-177.590,7.352,148.685
C06714=1164.966,233.024,-64.239,-177.594,7.349,148.685
C06715=1164.970,232.775,-64.213,-177.596,7.347,148.685
C06716=1164.975,232.527,-64.188,-177.599,7.344,148.685
C06717=1164.980,232.278,-64.162,-177.602,7.342,148.686
C06718=1164.984,232.029,-64.135,-177.604,7.340,148.686
C06719=1164.988,231.781,-64.110,-177.607,7.337,148.686
C06720=1164.992,231.532,-64.084,-177.610,7.334,148.686
C06721=1164.998,231.283,-64.058,-177.612,7.332,148.686
C06722=1165.002,231.035,-64.032,-177.615,7.329,148.686
C06723=1165.006,230.786,-64.006,-177.618,7.327,148.687
C06724=1165.010,230.538,-63.980,-177.620,7.324,148.687
C06725=1165.015,230.289,-63.954,-177.623,7.321,148.687
C06726=1165.020,230.040,-63.928,-177.626,7.319,148.687
C06727=1165.024,229.792,-63.902,-177.629,7.317,148.687
C06728=1165.028,229.543,-63.877,-177.631,7.314,148.687
C06729=1165.033,229.295,-63.851,-177.634,7.312,148.688
C06730=1165.037,229.046,-63.825,-177.637,7.309,148.688
C06731=1165.042,228.797,-63.800,-177.639,7.307,148.688
C06732=1165.046,228.549,-63.773,-177.642,7.304,148.688
C06733=1165.051,228.300,-63.747,-177.645,7.301,148.688
C06734=1165.055,228.052,-63.722,-177.648,7.299,148.689
C06735=1165.060,227.803,-63.696,-177.650,7.296,148.689
C06736=1165.064,227.554,-63.670,-177.653,7.294,148.689
C06737=1165.069,227.306,-63.645,-177.656,7.292,148.689
C06738=1165.073,227.057,-63.619,-177.659,7.289,148.689
C06739=1165.077,226.808,-63.593,-177.661,7.287,148.690
C06740=1165.082,226.560,-63.568,-177.664,7.284,148.690
C06741=1165.087,226.311,-63.541,-177.666,7.282,148.690
C06742=1165.091,226.062,-63.516,-177.669,7.279,148.690
C06743=1165.096,225.814,-63.491,-177.672,7.277,148.690
C06744=1165.100,225.565,-63.465,-177.674,7.274,148.690
C06745=1165.105,225.316,-63.439,-177.678,7.272,148.691
C06746=1165.110,225.068,-63.414,-177.680,7.269,148.691
C06747=1165.114,224.819,-63.388,-177.683,7.267,148.691
C06748=1165.118,224.570,-63.363,-177.685,7.265,148.691
C06749=1165.123,224.322,-63.337,-177.689,7.262,148.691
C06750=1165.127,224.073,-63.312,-177.691,7.260,148.691
C06751=1165.132,223.824,-63.286,-177.693,7.257,148.692
C06752=1165.136,223.576,-63.261,-177.697,7.254,148.692
C06753=1165.141,223.327,-63.235,-177.699,7.252,148.692
C06754=1165.145,223.078,-63.210,-177.702,7.250,148.692
C06755=1165.150,222.829,-63.185,-177.704,7.248,148.692
C06756=1165.154,222.581,-63.159,-177.707,7.245,148.692
C06757=1165.159,222.333,-63.134,-177.710,7.243,148.693
C06758=1165.163,222.084,-63.108,-177.713,7.240,148.693
C06759=1165.167,221.835,-63.084,-177.715,7.238,148.693
C06760=1165.172,221.587,-63.058,-177.718,7.235,148.693
C06761=1165.176,221.338,-63.032,-177.721,7.233,148.694
C06762=1165.181,221.089,-63.008,-177.723,7.231,148.694
C06763=1165.185,220.840,-62.982,-177.727,7.228,148.694
C06764=1165.190,220.592,-62.957,-177.729,7.226,148.694
C06765=1165.195,220.343,-62.932,-177.732,7.223,148.694
C06766=1165.199,220.094,-62.906,-177.734,7.221,148.695
C06767=1165.204,219.846,-62.880,-177.737,7.218,148.695
C06768=1165.208,219.597,-62.856,-177.740,7.216,148.695
C06769=1165.212,219.349,-62.831,-177.742,7.213,148.695
C06770=1165.217,219.099,-62.806,-177.745,7.212,148.695
C06771=1165.222,218.851,-62.780,-177.748,7.209,148.696
C06772=1165.226,218.602,-62.754,-177.751,7.207,148.696
C06773=1165.230,218.354,-62.730,-177.753,7.204,148.696
C06774=1165.235,218.105,-62.705,-177.756,7.202,148.696
C06775=1165.240,217.856,-62.680,-177.759,7.199,148.696
C06776=1165.244,217.607,-62.654,-177.761,7.197,148.697
C06777=1165.249,217.359,-62.630,-177.764,7.194,148.697
C06778=1165.253,217.110,-62.604,-177.766,7.192,148.697
C06779=1165.258,216.862,-62.580,-177.770,7.190,148.697
C06780=1165.262,216.613,-62.554,-177.772,7.187,148.697
C06781=1165.267,216.364,-62.529,-177.775,7.185,148.698
C06782=1165.271,216.116,-62.504,-177.778,7.182,148.698
C06783=1165.276,215.867,-62.479,-177.781,7.180,148.698
C06784=1165.280,215.617,-62.454,-177.783,7.177,148.698
C06785=1165.284,215.370,-62.430,-177.786,7.176,148.699
C06786=1165.289,215.120,-62.405,-177.789,7.173,148.699
C06787=1165.294,214.872,-62.379,-177.791,7.171,148.699
C06788=1165.298,214.623,-62.354,-177.794,7.169,148.699
C06789=1165.303,214.374,-62.330,-177.797,7.166,148.699
C06790=1165.307,214.125,-62.304,-177.799,7.164,148.700
C06791=1165.312,213.877,-62.280,-177.802,7.161,148.700
C06792=1165.316,213.628,-62.256,-177.805,7.159,148.700
C06793=1165.321,213.379,-62.231,-177.808,7.157,148.700
C06794=1165.325,213.131,-62.206,-177.810,7.155,148.700
C06795=1165.330,212.882,-62.181,-177.813,7.152,148.701
C06796=1165.335,212.633,-62.156,-177.815,7.150,148.701
C06797=1165.338,212.384,-62.131,-177.819,7.147,148.701
C06798=1165.343,212.136,-62.106,-177.821,7.145,148.701
C06799=1165.348,211.887,-62.082,-177.824,7.143,148.702
C06800=1165.352,211.638,-62.057,-177.827,7.141,148.702
C06801=1165.357,211.389,-62.032,-177.830,7.138,148.702
C06802=1165.361,211.141,-62.008,-177.832,7.136,148.702
C06803=1165.366,210.892,-61.983,-177.835,7.133,148.702
C06804=1165.370,210.644,-61.959,-177.838,7.131,148.703
C06805=1165.375,210.373,-61.931,-177.840,7.128,148.703
C06806=1165.380,210.102,-61.905,-177.844,7.126,148.703
C06807=1165.385,209.832,-61.878,-177.846,7.124,148.704
C06808=1165.390,209.561,-61.851,-177.849,7.121,148.704
C06809=1165.395,209.313,-61.826,-177.852,7.119,148.704
C06810=1165.399,209.064,-61.802,-177.855,7.116,148.704
C06811=1165.404,208.815,-61.777,-177.857,7.115,148.704
C06812=1165.408,208.566,-61.753,-177.860,7.112,148.705
C06813=1165.413,208.318,-61.728,-177.863,7.110,148.705
C06814=1165.417,208.069,-61.704,-177.866,7.107,148.705
C06815=1165.422,207.820,-61.679,-177.868,7.105,148.705
C06816=1165.427,207.571,-61.655,-177.871,7.103,148.706
C06817=1165.431,207.322,-61.630,-177.874,7.100,148.706
C06818=1165.436,207.074,-61.606,-177.877,7.098,148.706
C06819=1165.441,206.825,-61.581,-177.879,7.096,148.706
C06820=1165.445,206.577,-61.557,-177.882,7.094,148.706
C06821=1165.449,206.327,-61.533,-177.885,7.091,148.707
C06822=1165.454,206.079,-61.508,-177.887,7.089,148.707
C06823=1165.458,205.830,-61.484,-177.890,7.087,148.707
C06824=1165.463,205.581,-61.459,-177.893,7.085,148.707
C06825=1165.467,205.332,-61.435,-177.896,7.082,148.708
C06826=1165.472,205.083,-61.412,-177.898,7.080,148.708
C06827=1165.477,204.835,-61.387,-177.901,7.078,148.708
C06828=1165.482,204.586,-61.363,-177.904,7.075,148.708
C06829=1165.486,204.337,-61.338,-177.906,7.073,148.709
C06830=1165.491,204.088,-61.314,-177.909,7.071,148.709
C06831=1165.495,203.840,-61.290,-177.912,7.069,148.709
C06832=1165.500,203.591,-61.265,-177.914,7.067,148.709
C06833=1165.504,203.342,-61.241,-177.918,7.064,148.710
C06834=1165.509,203.093,-61.217,-177.920,7.062,148.710
C06835=1165.513,202.845,-61.193,-177.923,7.060,148.710
C06836=1165.518,202.596,-61.169,-177.925,7.057,148.710
C06837=1165.522,202.346,-61.145,-177.928,7.055,148.711
C06838=1165.527,202.098,-61.121,-177.931,7.053,148.711
C06839=1165.532,201.849,-61.096,-177.933,7.051,148.711
C06840=1165.536,201.601,-61.072,-177.937,7.048,148.711
C06841=1165.541,201.352,-61.049,-177.939,7.046,148.712
C06842=1165.545,201.103,-61.025,-177.942,7.044,148.712
C06843=1165.549,200.854,-61.000,-177.945,7.042,148.712
C06844=1165.554,200.605,-60.976,-177.947,7.040,148.712
C06845=1165.559,200.356,-60.952,-177.950,7.037,148.713
C06846=1165.563,200.108,-60.928,-177.952,7.035,148.713
C06847=1165.568,199.859,-60.905,-177.955,7.033,148.713
C06848=1165.573,199.610,-60.880,-177.958,7.031,148.713
C06849=1165.577,199.361,-60.856,-177.960,7.029,148.714
C06850=1165.582,199.112,-60.832,-177.964,7.026,148.714
C06851=1165.586,198.864,-60.808,-177.966,7.024,148.714
C06852=1165.591,198.615,-60.785,-177.969,7.022,148.714
C06853=1165.595,198.366,-60.761,-177.972,7.020,148.715
C06854=1165.600,198.117,-60.736,-177.975,7.018,148.715
C06855=1165.605,197.868,-60.713,-177.977,7.016,148.715
C06856=1165.609,197.620,-60.689,-177.980,7.013,148.716
C06857=1165.614,197.371,-60.665,-177.982,7.011,148.716
C06858=1165.618,197.122,-60.641,-177.985,7.008,148.716
C06859=1165.622,196.873,-60.618,-177.988,7.007,148.716
C06860=1165.627,196.624,-60.593,-177.990,7.004,148.716
C06861=1165.632,196.375,-60.570,-177.994,7.002,148.717
C06862=1165.636,196.127,-60.546,-177.996,7.000,148.717
C06863=1165.641,195.878,-60.522,-177.998,6.998,148.717
C06864=1165.646,195.629,-60.499,-178.002,6.995,148.718
C06865=1165.650,195.380,-60.475,-178.004,6.994,148.718
C06866=1165.655,195.131,-60.451,-178.007,6.992,148.718
C06867=1165.660,194.883,-60.427,-178.010,6.989,148.718
C06868=1165.664,194.634,-60.404,-178.012,6.987,148.719
C06869=1165.669,194.385,-60.380,-178.015,6.985,148.719
C06870=1165.673,194.136,-60.356,-178.018,6.982,148.719
C06871=1165.678,193.887,-60.333,-178.021,6.981,148.720
C06872=1165.683,193.638,-60.310,-178.023,6.979,148.720
C06873=1165.687,193.390,-60.286,-178.026,6.976,148.720
C06874=1165.692,193.141,-60.262,-178.029,6.974,148.720
C06875=1165.697,192.892,-60.239,-178.031,6.972,148.721
C06876=1165.701,192.643,-60.215,-178.034,6.970,148.721
C06877=1165.706,192.394,-60.191,-178.037,6.968,148.721
C06878=1165.710,192.145,-60.168,-178.040,6.966,148.722
C06879=1165.715,191.897,-60.144,-178.042,6.963,148.722
C06880=1165.719,191.648,-60.121,-178.045,6.961,148.722
C06881=1165.724,191.399,-60.097,-178.048,6.960,148.722
C06882=1165.729,191.150,-60.074,-178.050,6.957,148.722
C06883=1165.734,190.901,-60.051,-178.053,6.955,148.723
C06884=1165.737,190.653,-60.027,-178.056,6.953,148.723
C06885=1165.742,190.404,-60.004,-178.059,6.950,148.723
C06886=1165.747,190.155,-59.980,-178.061,6.948,148.724
C06887=1165.751,189.906,-59.957,-178.064,6.947,148.724
C06888=1165.756,189.657,-59.934,-178.067,6.944,148.724
C06889=1165.761,189.407,-59.910,-178.069,6.942,148.724
C06890=1165.765,189.159,-59.886,-178.072,6.940,148.725
C06891=1165.770,188.910,-59.863,-178.075,6.938,148.725
C06892=1165.774,188.661,-59.840,-178.078,6.935,148.725
C06893=1165.778,188.412,-59.817,-178.080,6.934,148.726
C06894=1165.783,188.163,-59.793,-178.083,6.932,148.726
C06895=1165.788,187.915,-59.770,-178.086,6.929,148.726
C06896=1165.793,187.666,-59.747,-178.088,6.927,148.726
C06897=1165.798,187.417,-59.724,-178.091,6.925,148.727
C06898=1165.802,187.168,-59.701,-178.094,6.923,148.727
C06899=1165.807,186.919,-59.678,-178.097,6.921,148.727
C06900=1165.811,186.670,-59.654,-178.099,6.919,148.728
C06901=1165.816,186.421,-59.631,-178.102,6.917,148.728
C06902=1165.821,186.172,-59.607,-178.105,6.915,148.728
C06903=1165.825,185.923,-59.585,-178.107,6.913,148.728
C06904=1165.830,185.675,-59.562,-178.110,6.911,148.729
C06905=1165.835,185.426,-59.538,-178.113,6.908,148.729
C06906=1165.839,185.177,-59.515,-178.116,6.906,148.730
C06907=1165.843,184.928,-59.492,-178.118,6.904,148.730
C06908=1165.848,184.679,-59.469,-178.121,6.903,148.730
C06909=1165.853,184.409,-59.444,-178.124,6.900,148.730
C06910=1165.858,184.140,-59.419,-178.127,6.897,148.731
C06911=1165.863,183.870,-59.394,-178.130,6.896,148.731
C06912=1165.868,183.600,-59.369,-178.133,6.893,148.731
C06913=1165.872,183.352,-59.347,-178.136,6.891,148.732
C06914=1165.877,183.103,-59.323,-178.138,6.889,148.732
C06915=1165.882,182.854,-59.300,-178.141,6.887,148.732
C06916=1165.886,182.606,-59.277,-178.144,6.885,148.733
C06917=1165.891,182.356,-59.255,-178.147,6.883,148.733
C06918=1165.896,182.107,-59.231,-178.149,6.881,148.733
C06919=1165.900,181.858,-59.209,-178.152,6.879,148.733
C06920=1165.905,181.610,-59.186,-178.155,6.877,148.734
C06921=1165.909,181.361,-59.163,-178.158,6.875,148.734
C06922=1165.914,181.111,-59.140,-178.160,6.873,148.734
C06923=1165.919,180.862,-59.117,-178.163,6.871,148.735
C06924=1165.923,180.614,-59.094,-178.166,6.868,148.735
C06925=1165.929,180.365,-59.072,-178.169,6.867,148.735
C06926=1165.933,180.116,-59.049,-178.171,6.865,148.736
C06927=1165.937,179.867,-59.026,-178.173,6.863,148.736
C06928=1165.941,179.618,-59.003,-178.177,6.860,148.736
C06929=1165.947,179.369,-58.981,-178.179,6.858,148.737
C06930=1165.952,179.120,-58.957,-178.182,6.857,148.737
C06931=1165.955,178.872,-58.935,-178.185,6.855,148.737
C06932=1165.961,178.623,-58.912,-178.188,6.852,148.737
C06933=1165.965,178.374,-58.890,-178.190,6.850,148.738
C06934=1165.970,178.124,-58.867,-178.193,6.848,148.738
C06935=1165.974,177.876,-58.844,-178.196,6.847,148.738
C06936=1165.979,177.627,-58.821,-178.198,6.845,148.739
C06937=1165.984,177.378,-58.799,-178.201,6.842,148.739
C06938=1165.988,177.129,-58.776,-178.204,6.840,148.739
C06939=1165.993,176.880,-58.754,-178.206,6.839,148.740
C06940=1165.998,176.631,-58.731,-178.209,6.837,148.740
C06941=1166.002,176.382,-58.709,-178.212,6.835,148.740
C06942=1166.007,176.133,-58.686,-178.215,6.832,148.741
C06943=1166.012,175.884,-58.664,-178.217,6.830,148.741
C06944=1166.016,175.635,-58.641,-178.220,6.829,148.741
C06945=1166.021,175.386,-58.619,-178.223,6.827,148.742
C06946=1166.025,175.138,-58.596,-178.226,6.824,148.742
C06947=1166.030,174.888,-58.573,-178.229,6.822,148.742
C06948=1166.035,174.640,-58.551,-178.231,6.820,148.742
C06949=1166.039,174.391,-58.529,-178.233,6.819,148.743
C06950=1166.044,174.141,-58.506,-178.236,6.817,148.743
C06951=1166.049,173.893,-58.484,-178.239,6.814,148.744
C06952=1166.054,173.643,-58.461,-178.242,6.813,148.744
C06953=1166.058,173.395,-58.438,-178.245,6.811,148.744
C06954=1166.062,173.146,-58.417,-178.247,6.809,148.744
C06955=1166.067,172.896,-58.394,-178.250,6.807,148.745
C06956=1166.072,172.648,-58.372,-178.252,6.805,148.745
C06957=1166.076,172.399,-58.350,-178.256,6.803,148.746
C06958=1166.081,172.149,-58.327,-178.258,6.801,148.746
C06959=1166.086,171.901,-58.304,-178.261,6.799,148.746
C06960=1166.090,171.652,-58.282,-178.263,6.797,148.746
C06961=1166.096,171.403,-58.260,-178.266,6.795,148.747
C06962=1166.100,171.154,-58.237,-178.269,6.793,148.747
C06963=1166.105,170.906,-58.216,-178.272,6.791,148.747
C06964=1166.110,170.656,-58.193,-178.275,6.789,148.748
C06965=1166.114,170.407,-58.171,-178.277,6.787,148.748
C06966=1166.118,170.159,-58.149,-178.280,6.786,148.749
C06967=1166.123,169.909,-58.127,-178.282,6.784,148.749
C06968=1166.128,169.660,-58.104,-178.285,6.781,148.749
C06969=1166.133,169.411,-58.082,-178.288,6.779,148.749
C06970=1166.137,169.162,-58.061,-178.291,6.777,148.750
C06971=1166.141,168.914,-58.038,-178.293,6.776,148.750
C06972=1166.147,168.665,-58.016,-178.296,6.774,148.751
C06973=1166.151,168.415,-57.993,-178.299,6.772,148.751
C06974=1166.156,168.167,-57.972,-178.302,6.770,148.751
C06975=1166.160,167.917,-57.950,-178.304,6.767,148.751
C06976=1166.165,167.669,-57.928,-178.307,6.766,148.752
C06977=1166.170,167.419,-57.905,-178.310,6.764,148.752
C06978=1166.175,167.171,-57.884,-178.312,6.762,148.753
C06979=1166.179,166.922,-57.861,-178.315,6.760,148.753
C06980=1166.184,166.673,-57.839,-178.318,6.759,148.753
C06981=1166.188,166.424,-57.817,-178.321,6.756,148.754
C06982=1166.193,166.175,-57.796,-178.324,6.754,148.754
C06983=1166.198,165.926,-57.773,-178.326,6.753,148.754
C06984=1166.203,165.677,-57.751,-178.329,6.751,148.754
C06985=1166.207,165.428,-57.729,-178.331,6.749,148.755
C06986=1166.212,165.179,-57.707,-178.334,6.747,148.755
C06987=1166.216,164.930,-57.685,-178.337,6.745,148.756
C06988=1166.221,164.681,-57.664,-178.339,6.744,148.756
C06989=1166.226,164.432,-57.642,-178.343,6.741,148.756
C06990=1166.230,164.183,-57.620,-178.345,6.739,148.757
C06991=1166.235,163.934,-57.598,-178.348,6.737,148.757
C06992=1166.240,163.685,-57.576,-178.351,6.736,148.757
C06993=1166.244,163.436,-57.555,-178.353,6.734,148.758
C06994=1166.249,163.187,-57.533,-178.356,6.732,148.758
C06995=1166.255,162.937,-57.511,-178.358,6.730,148.758
C06996=1166.259,162.688,-57.489,-178.361,6.728,148.759
C06997=1166.264,162.439,-57.467,-178.364,6.726,148.759
C06998=1166.269,162.191,-57.446,-178.367,6.724,148.759
C06999=1166.273,161.941,-57.424,-178.370,6.722,148.760
C07000=1166.278,161.693,-57.402,-178.372,6.721,148.760
C07001=1166.282,161.443,-57.380,-178.375,6.719,148.761
C07002=1166.287,161.194,-57.359,-178.378,6.717,148.761
C07003=1166.292,160.946,-57.337,-178.380,6.715,148.761
C07004=1166.296,160.696,-57.315,-178.383,6.714,148.762
C07005=1166.301,160.448,-57.293,-178.386,6.712,148.762
C07006=1166.305,160.199,-57.272,-178.389,6.710,148.762
C07007=1166.310,159.949,-57.251,-178.392,6.707,148.763
C07008=1166.315,159.701,-57.229,-178.395,6.706,148.763
C07009=1166.319,159.451,-57.207,-178.397,6.704,148.764
C07010=1166.324,159.203,-57.186,-178.399,6.702,148.764
C07011=1166.329,158.953,-57.165,-178.402,6.700,148.764
C07012=1166.333,158.704,-57.143,-178.405,6.698,148.764
C07013=1166.339,158.435,-57.120,-178.408,6.697,148.765
C07014=1166.344,158.167,-57.096,-178.411,6.694,148.765
C07015=1166.349,157.898,-57.073,-178.414,6.693,148.766
C07016=1166.354,157.629,-57.050,-178.417,6.691,148.766
C07017=1166.358,157.379,-57.028,-178.419,6.689,148.767
C07018=1166.364,157.130,-57.007,-178.422,6.687,148.767
C07019=1166.368,156.881,-56.985,-178.425,6.686,148.767
C07020=1166.373,156.633,-56.964,-178.428,6.683,148.768
C07021=1166.377,156.383,-56.943,-178.431,6.681,148.768
C07022=1166.382,156.134,-56.921,-178.433,6.680,148.768
C07023=1166.387,155.886,-56.900,-178.436,6.678,148.769
C07024=1166.391,155.636,-56.878,-178.439,6.676,148.769
C07025=1166.396,155.387,-56.856,-178.441,6.674,148.769
C07026=1166.401,155.138,-56.836,-178.444,6.672,148.770
C07027=1166.406,154.890,-56.814,-178.446,6.671,148.770
C07028=1166.410,154.640,-56.793,-178.449,6.669,148.770
C07029=1166.415,154.391,-56.771,-178.452,6.667,148.771
C07030=1166.420,154.142,-56.750,-178.454,6.665,148.771
C07031=1166.424,153.893,-56.729,-178.457,6.664,148.772
C07032=1166.429,153.643,-56.708,-178.460,6.662,148.772
C07033=1166.434,153.395,-56.686,-178.463,6.660,148.772
C07034=1166.439,153.145,-56.665,-178.465,6.658,148.773
C07035=1166.443,152.897,-56.644,-178.468,6.657,148.773
C07036=1166.448,152.648,-56.623,-178.471,6.655,148.773
C07037=1166.453,152.399,-56.601,-178.473,6.653,148.774
C07038=1166.458,152.149,-56.580,-178.477,6.651,148.774
C07039=1166.462,151.900,-56.560,-178.479,6.649,148.775
C07040=1166.467,151.652,-56.538,-178.482,6.647,148.775
C07041=1166.472,151.402,-56.517,-178.485,6.645,148.775
C07042=1166.476,151.153,-56.497,-178.487,6.644,148.776
C07043=1166.481,150.904,-56.475,-178.490,6.642,148.776
C07044=1166.486,150.655,-56.454,-178.493,6.640,148.776
C07045=1166.490,150.407,-56.433,-178.496,6.638,148.777
C07046=1166.495,150.157,-56.412,-178.498,6.637,148.777
C07047=1166.501,149.908,-56.391,-178.501,6.635,148.778
C07048=1166.504,149.658,-56.370,-178.504,6.633,148.778
C07049=1166.509,149.410,-56.348,-178.506,6.631,148.778
C07050=1166.514,149.161,-56.327,-178.509,6.630,148.779
C07051=1166.519,148.912,-56.307,-178.512,6.628,148.779
C07052=1166.524,148.663,-56.285,-178.514,6.626,148.780
C07053=1166.528,148.414,-56.265,-178.517,6.624,148.780
C07054=1166.533,148.165,-56.244,-178.520,6.623,148.780
C07055=1166.538,147.915,-56.223,-178.522,6.621,148.781
C07056=1166.542,147.666,-56.202,-178.525,6.619,148.781
C07057=1166.547,147.417,-56.181,-178.528,6.617,148.781
C07058=1166.552,147.168,-56.160,-178.531,6.616,148.782
C07059=1166.557,146.919,-56.139,-178.534,6.614,148.782
C07060=1166.561,146.670,-56.119,-178.536,6.613,148.783
C07061=1166.566,146.421,-56.098,-178.539,6.611,148.783
C07062=1166.571,146.172,-56.076,-178.542,6.609,148.784
C07063=1166.576,145.923,-56.056,-178.545,6.607,148.784
C07064=1166.581,145.674,-56.035,-178.547,6.606,148.784
C07065=1166.585,145.424,-56.014,-178.550,6.604,148.785
C07066=1166.590,145.175,-55.993,-178.553,6.602,148.785
C07067=1166.594,144.926,-55.973,-178.555,6.600,148.785
C07068=1166.600,144.677,-55.952,-178.558,6.599,148.786
C07069=1166.604,144.428,-55.932,-178.561,6.597,148.786
C07070=1166.609,144.179,-55.911,-178.563,6.595,148.787
C07071=1166.614,143.930,-55.890,-178.566,6.593,148.787
C07072=1166.618,143.681,-55.870,-178.569,6.592,148.787
C07073=1166.623,143.431,-55.849,-178.572,6.590,148.788
C07074=1166.628,143.182,-55.829,-178.574,6.588,148.788
C07075=1166.633,142.933,-55.808,-178.577,6.586,148.789
C07076=1166.637,142.684,-55.787,-178.580,6.585,148.789
C07077=1166.642,142.435,-55.766,-178.582,6.583,148.789
C07078=1166.647,142.186,-55.746,-178.585,6.581,148.790
C07079=1166.651,141.937,-55.726,-178.588,6.581,148.790
C07080=1166.657,141.688,-55.705,-178.590,6.579,148.791
C07081=1166.661,141.439,-55.684,-178.593,6.577,148.791
C07082=1166.666,141.190,-55.663,-178.596,6.575,148.791
C07083=1166.671,140.941,-55.643,-178.598,6.574,148.792
C07084=1166.675,140.692,-55.622,-178.601,6.572,148.792
C07085=1166.680,140.442,-55.601,-178.604,6.570,148.793
C07086=1166.685,140.194,-55.581,-178.607,6.569,148.793
C07087=1166.689,139.945,-55.561,-178.609,6.567,148.793
C07088=1166.694,139.695,-55.540,-178.612,6.565,148.794
C07089=1166.699,139.446,-55.520,-178.615,6.563,148.794
C07090=1166.703,139.197,-55.500,-178.617,6.562,148.795
C07091=1166.709,138.948,-55.479,-178.620,6.560,148.795
C07092=1166.713,138.699,-55.458,-178.623,6.558,148.796
C07093=1166.717,138.450,-55.438,-178.626,6.557,148.796
C07094=1166.723,138.200,-55.417,-178.629,6.555,148.796
C07095=1166.727,137.951,-55.397,-178.631,6.553,148.797
C07096=1166.732,137.702,-55.377,-178.634,6.552,148.797
C07097=1166.736,137.453,-55.357,-178.637,6.550,148.798
C07098=1166.742,137.204,-55.336,-178.639,6.549,148.798
C07099=1166.747,136.955,-55.316,-178.642,6.547,148.798
C07100=1166.751,136.706,-55.296,-178.644,6.545,148.799
C07101=1166.756,136.457,-55.276,-178.647,6.544,148.799
C07102=1166.761,136.208,-55.255,-178.650,6.542,148.799
C07103=1166.766,135.958,-55.235,-178.653,6.541,148.800
C07104=1166.770,135.709,-55.215,-178.656,6.539,148.800
C07105=1166.774,135.460,-55.194,-178.658,6.537,148.801
C07106=1166.780,135.210,-55.174,-178.661,6.535,148.801
C07107=1166.784,134.961,-55.154,-178.664,6.534,148.802
C07108=1166.789,134.713,-55.134,-178.666,6.532,148.802
C07109=1166.794,134.464,-55.114,-178.669,6.530,148.802
C07110=1166.799,134.215,-55.094,-178.671,6.529,148.803
C07111=1166.804,133.965,-55.073,-178.674,6.528,148.803
C07112=1166.808,133.716,-55.053,-178.677,6.526,148.804
C07113=1166.813,133.467,-55.033,-178.680,6.524,148.804
C07114=1166.818,133.217,-55.013,-178.683,6.523,148.805
C07115=1166.823,132.969,-54.993,-178.685,6.521,148.805
C07116=1166.827,132.719,-54.973,-178.688,6.519,148.805
C07117=1166.833,132.451,-54.951,-178.691,6.517,148.806
C07118=1166.838,132.182,-54.930,-178.694,6.516,148.806
C07119=1166.843,131.913,-54.908,-178.697,6.514,148.807
C07120=1166.848,131.645,-54.886,-178.699,6.513,148.807
C07121=1166.853,131.396,-54.867,-178.702,6.511,148.808
C07122=1166.857,131.147,-54.846,-178.705,6.510,148.808
C07123=1166.862,130.897,-54.827,-178.708,6.508,148.809
C07124=1166.867,130.649,-54.807,-178.711,6.506,148.809
C07125=1166.872,130.399,-54.786,-178.713,6.504,148.809
C07126=1166.877,130.150,-54.766,-178.716,6.503,148.810
C07127=1166.882,129.901,-54.746,-178.719,6.501,148.810
C07128=1166.886,129.651,-54.727,-178.721,6.500,148.811
C07129=1166.891,129.403,-54.707,-178.724,6.499,148.811
C07130=1166.896,129.153,-54.687,-178.727,6.497,148.812
C07131=1166.901,128.904,-54.667,-178.729,6.495,148.812
C07132=1166.905,128.655,-54.647,-178.732,6.493,148.812
C07133=1166.911,128.406,-54.628,-178.735,6.492,148.813
C07134=1166.915,128.157,-54.607,-178.738,6.490,148.813
C07135=1166.920,127.907,-54.588,-178.740,6.488,148.814
C07136=1166.925,127.658,-54.568,-178.743,6.488,148.814
C07137=1166.930,127.410,-54.548,-178.746,6.486,148.815
C07138=1166.934,127.160,-54.528,-178.748,6.484,148.815
C07139=1166.939,126.910,-54.509,-178.751,6.482,148.815
C07140=1166.944,126.662,-54.489,-178.754,6.481,148.816
C07141=1166.949,126.413,-54.469,-178.756,6.479,148.816
C07142=1166.954,126.163,-54.449,-178.760,6.478,148.817
C07143=1166.957,125.914,-54.430,-178.762,6.477,148.817
C07144=1166.963,125.666,-54.410,-178.764,6.475,148.818
C07145=1166.967,125.416,-54.391,-178.767,6.473,148.818
C07146=1166.972,125.166,-54.371,-178.770,6.472,148.818
C07147=1166.977,124.918,-54.351,-178.773,6.470,148.819
C07148=1166.982,124.669,-54.331,-178.776,6.468,148.819
C07149=1166.987,124.419,-54.312,-178.778,6.468,148.820
C07150=1166.992,124.170,-54.292,-178.781,6.466,148.820
C07151=1166.997,123.921,-54.273,-178.783,6.464,148.821
C07152=1167.000,123.672,-54.253,-178.786,6.462,148.821
C07153=1167.006,123.423,-54.234,-178.789,6.461,148.821
C07154=1167.011,123.174,-54.214,-178.792,6.459,148.822
C07155=1167.015,122.924,-54.194,-178.794,6.458,148.822
C07156=1167.021,122.675,-54.175,-178.797,6.457,148.823
C07157=1167.025,122.426,-54.155,-178.799,6.455,148.823
C07158=1167.030,122.176,-54.136,-178.802,6.453,148.824
C07159=1167.035,121.927,-54.117,-178.805,6.452,148.824
C07160=1167.039,121.678,-54.097,-178.808,6.450,148.825
C07161=1167.044,121.429,-54.077,-178.810,6.449,148.825
C07162=1167.049,121.180,-54.058,-178.813,6.447,148.825
C07163=1167.054,120.930,-54.038,-178.816,6.446,148.826
C07164=1167.059,120.682,-54.019,-178.819,6.444,148.826
C07165=1167.063,120.432,-54.000,-178.821,6.443,148.827
C07166=1167.068,120.183,-53.980,-178.824,6.442,148.827
C07167=1167.073,119.934,-53.961,-178.826,6.440,148.828
C07168=1167.077,119.685,-53.942,-178.829,6.438,148.828
C07169=1167.083,119.436,-53.922,-178.832,6.437,148.829
C07170=1167.088,119.186,-53.903,-178.835,6.435,148.829
C07171=1167.092,118.937,-53.883,-178.837,6.434,148.830
C07172=1167.097,118.688,-53.864,-178.840,6.433,148.830
C07173=1167.102,118.439,-53.845,-178.843,6.431,148.830
C07174=1167.107,118.190,-53.826,-178.846,6.430,148.831
C07175=1167.111,117.940,-53.806,-178.848,6.428,148.831
C07176=1167.117,117.691,-53.788,-178.851,6.427,148.832
C07177=1167.121,117.441,-53.768,-178.853,6.425,148.832
C07178=1167.127,117.192,-53.749,-178.856,6.424,148.833
C07179=1167.131,116.943,-53.730,-178.859,6.422,148.833
C07180=1167.135,116.694,-53.710,-178.862,6.420,148.834
C07181=1167.141,116.445,-53.691,-178.864,6.419,148.834
C07182=1167.145,116.196,-53.672,-178.867,6.418,148.834
C07183=1167.150,115.947,-53.653,-178.870,6.416,148.835
C07184=1167.154,115.697,-53.634,-178.873,6.415,148.835
C07185=1167.160,115.448,-53.615,-178.875,6.414,148.836
C07186=1167.165,115.198,-53.595,-178.877,6.412,148.836
C07187=1167.169,114.950,-53.577,-178.881,6.411,148.837
C07188=1167.174,114.700,-53.557,-178.883,6.409,148.837
C07189=1167.180,114.451,-53.538,-178.886,6.407,148.838
C07190=1167.184,114.201,-53.519,-178.888,6.406,148.838
C07191=1167.189,113.953,-53.500,-178.891,6.405,148.839
C07192=1167.193,113.703,-53.481,-178.894,6.403,148.839
C07193=1167.199,113.454,-53.462,-178.897,6.402,148.840
C07194=1167.204,113.205,-53.443,-178.899,6.401,148.840
C07195=1167.208,112.956,-53.424,-178.902,6.399,148.840
C07196=1167.213,112.707,-53.405,-178.905,6.398,148.841
C07197=1167.218,112.457,-53.386,-178.908,6.396,148.841
C07198=1167.223,112.208,-53.367,-178.910,6.395,148.842
C07199=1167.227,111.959,-53.348,-178.912,6.393,148.842
C07200=1167.233,111.709,-53.329,-178.916,6.392,148.843
C07201=1167.237,111.460,-53.310,-178.918,6.390,148.843
C07202=1167.242,111.211,-53.291,-178.920,6.389,148.844
C07203=1167.247,110.962,-53.273,-178.923,6.387,148.844
C07204=1167.252,110.713,-53.253,-178.926,6.386,148.845
C07205=1167.256,110.463,-53.236,-178.929,6.384,148.845
C07206=1167.261,110.214,-53.216,-178.931,6.384,148.846
C07207=1167.266,109.965,-53.197,-178.934,6.382,148.846
C07208=1167.271,109.715,-53.178,-178.937,6.380,148.847
C07209=1167.275,109.466,-53.160,-178.940,6.379,148.847
C07210=1167.281,109.217,-53.141,-178.942,6.378,148.847
C07211=1167.285,108.968,-53.122,-178.945,6.376,148.848
C07212=1167.290,108.719,-53.103,-178.948,6.375,148.848
C07213=1167.295,108.469,-53.084,-178.951,6.373,148.849
C07214=1167.299,108.220,-53.066,-178.953,6.372,148.849
C07215=1167.305,107.971,-53.047,-178.956,6.371,148.850
C07216=1167.309,107.722,-53.028,-178.959,6.369,148.850
C07217=1167.315,107.472,-53.009,-178.961,6.368,148.851
C07218=1167.319,107.224,-52.991,-178.964,6.366,148.851
C07219=1167.324,106.974,-52.972,-178.967,6.365,148.852
C07220=1167.329,106.724,-52.954,-178.969,6.363,148.852
C07221=1167.334,106.457,-52.934,-178.972,6.362,148.853
C07222=1167.339,106.187,-52.913,-178.975,6.361,148.853
C07223=1167.344,105.919,-52.894,-178.978,6.359,148.854
C07224=1167.350,105.651,-52.873,-178.981,6.358,148.854
C07225=1167.355,105.402,-52.855,-178.983,6.356,148.855
C07226=1167.359,105.152,-52.835,-178.986,6.355,148.855
C07227=1167.364,104.903,-52.817,-178.989,6.354,148.856
C07228=1167.369,104.654,-52.799,-178.991,6.352,148.856
C07229=1167.374,104.405,-52.780,-178.994,6.351,148.857
C07230=1167.379,104.155,-52.762,-178.997,6.350,148.857
C07231=1167.384,103.906,-52.744,-179.000,6.348,148.858
C07232=1167.388,103.657,-52.725,-179.002,6.347,148.858
C07233=1167.394,103.407,-52.706,-179.005,6.345,148.858
C07234=1167.398,103.158,-52.688,-179.008,6.344,148.859
C07235=1167.403,102.910,-52.670,-179.010,6.343,148.859
C07236=1167.408,102.659,-52.651,-179.013,6.341,148.860
C07237=1167.413,102.410,-52.633,-179.016,6.340,148.861
C07238=1167.418,102.162,-52.614,-179.018,6.339,148.861
C07239=1167.422,101.912,-52.596,-179.021,6.337,148.861
C07240=1167.428,101.662,-52.577,-179.024,6.337,148.862
C07241=1167.432,101.413,-52.559,-179.026,6.335,148.862
C07242=1167.437,101.165,-52.540,-179.029,6.333,148.863
C07243=1167.441,100.915,-52.522,-179.031,6.332,148.863
C07244=1167.446,100.666,-52.504,-179.034,6.331,148.864
C07245=1167.452,100.416,-52.485,-179.037,6.329,148.864
C07246=1167.457,100.167,-52.467,-179.039,6.328,148.865
C07247=1167.461,99.918,-52.449,-179.043,6.327,148.865
C07248=1167.466,99.669,-52.430,-179.045,6.325,148.866
C07249=1167.471,99.419,-52.412,-179.047,6.324,148.866
C07250=1167.476,99.170,-52.394,-179.051,6.323,148.867
C07251=1167.481,98.921,-52.376,-179.053,6.321,148.867
C07252=1167.486,98.671,-52.358,-179.055,6.320,148.868
C07253=1167.490,98.422,-52.340,-179.059,6.319,148.868
C07254=1167.495,98.173,-52.321,-179.061,6.317,148.869
C07255=1167.500,97.924,-52.303,-179.064,6.316,148.869
C07256=1167.505,97.675,-52.285,-179.067,6.315,148.870
C07257=1167.511,97.425,-52.266,-179.069,6.313,148.870
C07258=1167.515,97.175,-52.248,-179.072,6.312,148.871
C07259=1167.520,96.926,-52.230,-179.075,6.311,148.871
C07260=1167.525,96.677,-52.212,-179.078,6.309,148.872
C07261=1167.530,96.428,-52.194,-179.080,6.308,148.872
C07262=1167.535,96.179,-52.176,-179.083,6.307,148.873
C07263=1167.539,95.929,-52.158,-179.086,6.305,148.873
C07264=1167.544,95.680,-52.140,-179.088,6.305,148.874
C07265=1167.549,95.430,-52.122,-179.091,6.303,148.874
C07266=1167.554,95.181,-52.104,-179.093,6.302,148.875
C07267=1167.558,94.932,-52.086,-179.096,6.301,148.875
C07268=1167.563,94.683,-52.068,-179.099,6.299,148.876
C07269=1167.569,94.433,-52.049,-179.101,6.298,148.876
C07270=1167.574,94.184,-52.031,-179.104,6.297,148.876
C07271=1167.578,93.934,-52.013,-179.107,6.295,148.877
C07272=1167.583,93.685,-51.995,-179.109,6.294,148.878
C07273=1167.588,93.436,-51.977,-179.112,6.293,148.878
C07274=1167.593,93.187,-51.959,-179.115,6.292,148.879
C07275=1167.598,92.937,-51.942,-179.117,6.290,148.879
C07276=1167.603,92.688,-51.924,-179.120,6.289,148.879
C07277=1167.608,92.439,-51.906,-179.123,6.288,148.880
C07278=1167.613,92.190,-51.888,-179.125,6.287,148.880
C07279=1167.617,91.941,-51.870,-179.128,6.285,148.881
C07280=1167.622,91.691,-51.852,-179.131,6.284,148.882
C07281=1167.627,91.442,-51.834,-179.133,6.283,148.882
C07282=1167.632,91.192,-51.817,-179.136,6.282,148.882
C07283=1167.636,90.943,-51.799,-179.139,6.280,148.883
C07284=1167.641,90.693,-51.781,-179.141,6.279,148.883
C07285=1167.646,90.444,-51.763,-179.144,6.278,148.884
C07286=1167.651,90.195,-51.745,-179.147,6.276,148.885
C07287=1167.656,89.945,-51.728,-179.149,6.276,148.885
C07288=1167.661,89.696,-51.710,-179.152,6.274,148.886
C07289=1167.666,89.447,-51.692,-179.155,6.273,148.886
C07290=1167.671,89.198,-51.674,-179.157,6.272,148.886
C07291=1167.676,88.948,-51.656,-179.160,6.270,148.887
C07292=1167.681,88.699,-51.639,-179.162,6.269,148.888
C07293=1167.685,88.450,-51.621,-179.165,6.268,148.888
C07294=1167.690,88.201,-51.603,-179.168,6.266,148.889
C07295=1167.696,87.951,-51.586,-179.170,6.265,148.889
C07296=1167.701,87.702,-51.568,-179.174,6.264,148.890
C07297=1167.705,87.453,-51.550,-179.176,6.263,148.890
C07298=1167.711,87.203,-51.533,-179.179,6.262,148.890
C07299=1167.715,86.954,-51.515,-179.182,6.260,148.891
C07300=1167.720,86.705,-51.497,-179.184,6.259,148.892
C07301=1167.725,86.455,-51.480,-179.187,6.258,148.892
C07302=1167.730,86.206,-51.462,-179.189,6.257,148.893
C07303=1167.735,85.957,-51.444,-179.192,6.255,148.893
